KUKA KRL program: MyProgram_300().src

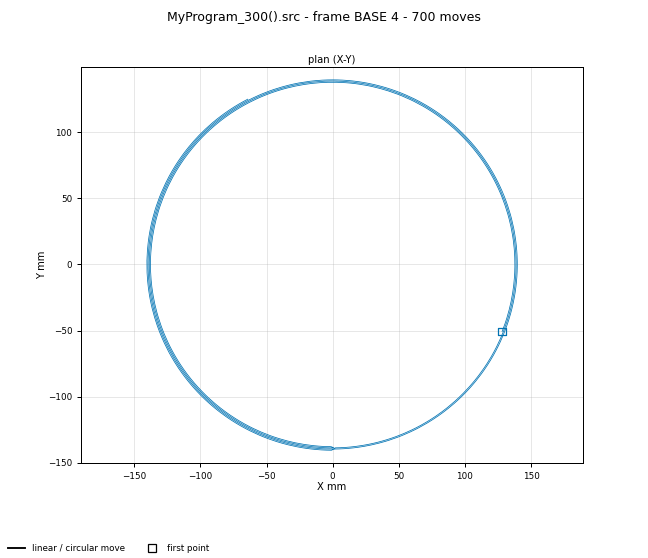
[picture p0: tool path of MyProgram_300().src in frame BASE 4, 700 of 700 moves have a stored position in this frame; points joined in program order, loops and branches not executed]
&ACCESS RVP
&REL 1
&PARAM TEMPLATE = C:\KRC\Roboter\Template\vorgabe
&PARAM EDITMASK = *
DEF MyProgram_300()
; ---- Setting reference (Base) ----
$BASE = BASE_DATA[4]

; --------------------------
; ---- Setting tool (TCP) ----
$TOOL = TOOL_DATA[3]
; --------------------------

$VEL.CP = VEL_APROX_PRINT
Startdeposition()
$VEL.CP = VEL_PRINT
LIN {X 128.1202,Y -50.7216,Z 179,A -18.2901,B 5.6421,C 0.2906,E1 5.7988,E2 470.655} C_DIS
LIN {X 129.3366,Y -47.5343,Z 179,A -16.9067,B 5.6423,C 0.2873,E1 5.8002,E2 469.2749} C_DIS
LIN {X 130.4678,Y -44.3354,Z 179,A -15.4081,B 5.6425,C 0.2821,E1 5.8015,E2 467.7637} C_DIS
LIN {X 131.6398,Y -40.7171,Z 179,A -13.99,B 5.6426,C 0.2803,E1 5.8027,E2 466.3653} C_DIS
LIN {X 132.591,Y -37.5041,Z 179,A -12.6322,B 5.6428,C 0.277,E1 5.8038,E2 465.0108} C_DIS
LIN {X 133.4585,Y -34.2894,Z 179,A -11.2835,B 5.643,C 0.2738,E1 5.8047,E2 463.6656} C_DIS
LIN {X 134.2751,Y -30.9365,Z 179,A -9.9543,B 5.643,C 0.2714,E1 5.8056,E2 462.3488} C_DIS
LIN {X 134.922,Y -27.9842,Z 179,A -8.7683,B 5.6432,C 0.269,E1 5.8063,E2 461.1708} C_DIS
LIN {X 135.5678,Y -24.6646,Z 179,A -7.2924,B 5.6434,C 0.264,E1 5.807,E2 459.6847} C_DIS
LIN {X 136.1099,Y -21.4723,Z 179,A -5.9815,B 5.6436,C 0.2607,E1 5.8076,E2 458.3773} C_DIS
LIN {X 136.5737,Y -18.2924,Z 179,A -4.6235,B 5.6438,C 0.2566,E1 5.8081,E2 457.0154} C_DIS
LIN {X 136.9237,Y -15.4683,Z 179,A -3.4321,B 5.6439,C 0.2531,E1 5.8085,E2 455.8221} C_DIS
LIN {X 137.2715,Y -11.9803,Z 179,A -2.254,B 5.6439,C 0.2533,E1 5.8088,E2 454.6786} C_DIS
LIN {X 137.5087,Y -8.8529,Z 179,A -0.9837,B 5.644,C 0.2502,E1 5.8091,E2 453.4116} C_DIS
LIN {X 137.658,Y -6.1429,Z 179,A 0.3699,B 5.6443,C 0.2434,E1 5.8093,E2 452.0283} C_DIS
LIN {X 137.7866,Y -1.5259,Z 179,A 2.0898,B 5.6444,C 0.2411,E1 5.8093,E2 450.3327} C_DIS
LIN {X 137.78,Y 1.9181,Z 179,A 3.3831,B 5.6445,C 0.2392,E1 5.8093,E2 449.056} C_DIS
LIN {X 137.7029,Y 4.993,Z 179,A 4.7743,B 5.6447,C 0.2338,E1 5.8093,E2 447.6496} C_DIS
LIN {X 137.58,Y 7.6943,Z 179,A 5.9871,B 5.6449,C 0.2292,E1 5.8091,E2 446.4246} C_DIS
LIN {X 137.2376,Y 12.3815,Z 179,A 7.8975,B 5.6451,C 0.2243,E1 5.8086,E2 444.5183} C_DIS
LIN {X 136.8687,Y 15.9359,Z 179,A 9.0863,B 5.6451,C 0.2248,E1 5.8083,E2 443.3665} C_DIS
LIN {X 136.5205,Y 18.6981,Z 179,A 10.364,B 5.6453,C 0.2196,E1 5.8078,E2 442.0727} C_DIS
LIN {X 136.0468,Y 21.8798,Z 179,A 11.6707,B 5.6454,C 0.2163,E1 5.8072,E2 440.7691} C_DIS
LIN {X 135.3992,Y 25.5723,Z 179,A 13.1704,B 5.6456,C 0.2129,E1 5.8065,E2 439.2758} C_DIS
LIN {X 134.7738,Y 28.6874,Z 179,A 14.4849,B 5.6457,C 0.2093,E1 5.8058,E2 437.9612} C_DIS
LIN {X 134.1493,Y 31.4869,Z 179,A 15.65,B 5.6458,C 0.2064,E1 5.805,E2 436.7989} C_DIS
LIN {X 133.3541,Y 34.7007,Z 179,A 17.1029,B 5.646,C 0.2014,E1 5.804,E2 435.3355} C_DIS
LIN {X 132.3654,Y 38.2933,Z 179,A 18.5158,B 5.646,C 0.1993,E1 5.803,E2 433.9389} C_DIS
LIN {X 131.3361,Y 41.6851,Z 179,A 19.9227,B 5.6462,C 0.1963,E1 5.8018,E2 432.5396} C_DIS
LIN {X 130.3079,Y 44.7966,Z 179,A 21.268,B 5.6462,C 0.1929,E1 5.8006,E2 431.1958} C_DIS
LIN {X 129.1837,Y 47.9425,Z 179,A 22.6404,B 5.6464,C 0.1895,E1 5.7993,E2 429.8246} C_DIS
LIN {X 127.9564,Y 51.1281,Z 179,A 24.0286,B 5.6465,C 0.1862,E1 5.7979,E2 428.4397} C_DIS
LIN {X 126.6436,Y 54.2982,Z 179,A 25.2652,B 5.6465,C 0.1854,E1 5.7966,E2 427.2263} C_DIS
LIN {X 125.23,Y 57.4833,Z 179,A 26.8315,B 5.6467,C 0.1798,E1 5.7948,E2 425.6445} C_DIS
LIN {X 123.762,Y 60.5793,Z 179,A 28.0749,B 5.6467,C 0.1789,E1 5.7933,E2 424.4233} C_DIS
LIN {X 122.1657,Y 63.7367,Z 179,A 29.6872,B 5.6469,C 0.173,E1 5.7912,E2 422.7925} C_DIS
LIN {X 120.2258,Y 67.3282,Z 179,A 31.3362,B 5.647,C 0.1695,E1 5.789,E2 421.1488} C_DIS
LIN {X 118.2543,Y 70.7336,Z 179,A 33.0192,B 5.6472,C 0.1648,E1 5.7866,E2 419.4592} C_DIS
LIN {X 115.8832,Y 74.555,Z 179,A 34.7836,B 5.6472,C 0.1619,E1 5.784,E2 417.7075} C_DIS
LIN {X 113.7346,Y 77.793,Z 179,A 36.4307,B 5.6474,C 0.1576,E1 5.7814,E2 416.0558} C_DIS
LIN {X 111.1958,Y 81.3807,Z 179,A 38.1794,B 5.6474,C 0.1546,E1 5.7786,E2 414.3164} C_DIS
LIN {X 108.6384,Y 84.7654,Z 179,A 39.9277,B 5.6476,C 0.1508,E1 5.7756,E2 412.5695} C_DIS
LIN {X 105.9924,Y 88.0508,Z 179,A 41.621,B 5.6476,C 0.1478,E1 5.7726,E2 410.8833} C_DIS
LIN {X 103.1924,Y 91.316,Z 179,A 43.4004,B 5.6477,C 0.1441,E1 5.7694,E2 409.1045} C_DIS
LIN {X 100.537,Y 94.2325,Z 179,A 45.056,B 5.6478,C 0.1404,E1 5.7662,E2 407.4466} C_DIS
LIN {X 97.4358,Y 97.4358,Z 179,A 46.8335,B 5.6478,C 0.1378,E1 5.7627,E2 405.6782} C_DIS
LIN {X 94.6416,Y 100.1512,Z 179,A 48.4576,B 5.648,C 0.1345,E1 5.7595,E2 404.0533} C_DIS
LIN {X 91.5999,Y 102.9413,Z 179,A 50.153,B 5.648,C 0.1315,E1 5.7559,E2 402.3603} C_DIS
LIN {X 88.2261,Y 105.8471,Z 179,A 51.9951,B 5.6481,C 0.1282,E1 5.752,E2 400.519} C_DIS
LIN {X 84.7654,Y 108.6384,Z 179,A 53.6964,B 5.6481,C 0.127,E1 5.7483,E2 398.836} C_DIS
LIN {X 81.5672,Y 111.0588,Z 179,A 55.3993,B 5.6482,C 0.1236,E1 5.7445,E2 397.1285} C_DIS
LIN {X 78.3355,Y 113.3623,Z 179,A 57.0178,B 5.6482,C 0.1214,E1 5.7408,E2 395.5139} C_DIS
LIN {X 74.8523,Y 115.6912,Z 179,A 58.7505,B 5.6483,C 0.1187,E1 5.7368,E2 393.7822} C_DIS
LIN {X 71.1191,Y 118.0229,Z 179,A 60.5116,B 5.6483,C 0.1169,E1 5.7326,E2 392.0298} C_DIS
LIN {X 67.896,Y 119.9067,Z 179,A 62.1383,B 5.6484,C 0.1137,E1 5.7286,E2 390.3937} C_DIS
LIN {X 64.437,Y 121.798,Z 179,A 63.6331,B 5.6484,C 0.1134,E1 5.725,E2 388.917} C_DIS
LIN {X 61.589,Y 123.2639,Z 179,A 64.888,B 5.6484,C 0.1127,E1 5.7219,E2 387.6718} C_DIS
LIN {X 58.6174,Y 124.7055,Z 179,A 66.4336,B 5.6485,C 0.1087,E1 5.718,E2 386.1049} C_DIS
LIN {X 54.9717,Y 126.3524,Z 179,A 67.7497,B 5.6485,C 0.1114,E1 5.7147,E2 384.832} C_DIS
LIN {X 52.3099,Y 127.48,Z 179,A 69.1382,B 5.6485,C 0.1075,E1 5.7111,E2 383.4206} C_DIS
LIN {X 49.1296,Y 128.7391,Z 179,A 70.6713,B 5.6486,C 0.1045,E1 5.707,E2 381.8739} C_DIS
LIN {X 45.4349,Y 130.0866,Z 179,A 71.9702,B 5.6486,C 0.1074,E1 5.7037,E2 380.6169} C_DIS
LIN {X 42.322,Y 131.1327,Z 179,A 73.5162,B 5.6486,C 0.1037,E1 5.6996,E2 379.0489} C_DIS
LIN {X 39.111,Y 132.1259,Z 179,A 74.9014,B 5.6486,C 0.1027,E1 5.6959,E2 377.6655} C_DIS
LIN {X 35.8968,Y 133.0352,Z 179,A 76.3077,B 5.6486,C 0.1014,E1 5.6921,E2 376.2573} C_DIS
LIN {X 32.6824,Y 133.8612,Z 179,A 77.4929,B 5.6486,C 0.1029,E1 5.6889,E2 375.0966} C_DIS
LIN {X 29.8812,Y 134.5161,Z 179,A 78.8355,B 5.6486,C 0.1002,E1 5.6852,E2 373.7363} C_DIS
LIN {X 26.6742,Y 135.1886,Z 179,A 80.3098,B 5.6487,C 0.098,E1 5.6812,E2 372.2485} C_DIS
LIN {X 22.9157,Y 135.874,Z 179,A 81.7673,B 5.6487,C 0.0988,E1 5.6772,E2 370.8077} C_DIS
LIN {X 19.8806,Y 136.3515,Z 179,A 83.0363,B 5.6487,C 0.0983,E1 5.6737,E2 369.5401} C_DIS
LIN {X 17.1127,Y 136.7283,Z 179,A 84.1924,B 5.6487,C 0.098,E1 5.6705,E2 368.3851} C_DIS
LIN {X 13.5516,Y 137.1253,Z 179,A 85.6745,B 5.6487,C 0.0975,E1 5.6664,E2 366.9045} C_DIS
LIN {X 10.1212,Y 137.4206,Z 179,A 87.0261,B 5.6487,C 0.0982,E1 5.6626,E2 365.5633} C_DIS
LIN {X 6.1429,Y 137.658,Z 179,A 88.8676,B 5.6487,C 0.0956,E1 5.6574,E2 363.6997} C_DIS
LIN {X 3.0585,Y 137.7611,Z 179,A 90.0316,B 5.6487,C 0.0969,E1 5.6542,E2 362.551} C_DIS
LIN {X -0.3905,Y 137.7929,Z 179,A 91.4644,B 5.6487,C 0.0969,E1 5.6502,E2 361.119} C_DIS
LIN {X -3.7662,Y 137.7414,Z 179,A 92.7926,B 5.6487,C 0.0978,E1 5.6466,E2 359.8007} C_DIS
LIN {X -6.5399,Y 137.6381,Z 179,A 93.8803,B 5.6487,C 0.0987,E1 5.6435,E2 358.7218} C_DIS
LIN {X -9.6512,Y 137.4549,Z 179,A 95.1792,B 5.6487,C 0.0989,E1 5.6399,E2 357.4232} C_DIS
LIN {X -12.9748,Y 137.1807,Z 179,A 96.6705,B 5.6487,C 0.0979,E1 5.6357,E2 355.9197} C_DIS
LIN {X -15.9359,Y 136.8687,Z 179,A 97.8121,B 5.6487,C 0.0994,E1 5.6326,E2 354.7906} C_DIS
LIN {X -19.278,Y 136.4376,Z 179,A 99.1541,B 5.6487,C 0.1006,E1 5.6289,E2 353.4567} C_DIS
LIN {X -21.8798,Y 136.0468,Z 179,A 100.4719,B 5.6487,C 0.0984,E1 5.6252,E2 352.112} C_DIS
LIN {X -25.4832,Y 135.4163,Z 179,A 102.0026,B 5.6487,C 0.099,E1 5.621,E2 350.5809} C_DIS
LIN {X -28.6874,Y 134.7738,Z 179,A 103.3702,B 5.6487,C 0.0996,E1 5.6172,E2 349.213} C_DIS
LIN {X -31.9883,Y 134.0285,Z 179,A 104.784,B 5.6487,C 0.1004,E1 5.6134,E2 347.7993} C_DIS
LIN {X -35.0817,Y 133.2525,Z 179,A 105.9762,B 5.6487,C 0.1028,E1 5.6102,E2 346.6243} C_DIS
LIN {X -37.9154,Y 132.476,Z 179,A 107.3552,B 5.6487,C 0.1019,E1 5.6065,E2 345.2268} C_DIS
LIN {X -41.3051,Y 131.4575,Z 179,A 108.9235,B 5.6487,C 0.102,E1 5.6022,E2 343.6474} C_DIS
LIN {X -44.745,Y 130.3258,Z 179,A 110.3596,B 5.6487,C 0.1041,E1 5.5985,E2 342.2209} C_DIS
LIN {X -47.9425,Y 129.1837,Z 179,A 111.7853,B 5.6486,C 0.1053,E1 5.5947,E2 340.7945} C_DIS
LIN {X -51.1281,Y 127.9564,Z 179,A 113.2197,B 5.6486,C 0.1066,E1 5.591,E2 339.3592} C_DIS
LIN {X -54.2982,Y 126.6436,Z 179,A 114.4971,B 5.6486,C 0.1098,E1 5.5878,E2 338.1013} C_DIS
LIN {X -57.4498,Y 125.2455,Z 179,A 116.1123,B 5.6486,C 0.1094,E1 5.5836,E2 336.4647} C_DIS
LIN {X -60.5793,Y 123.762,Z 179,A 117.4029,B 5.6484,C 0.1128,E1 5.5804,E2 335.1935} C_DIS
LIN {X -63.2885,Y 122.4011,Z 179,A 118.9792,B 5.6484,C 0.111,E1 5.5764,E2 333.5792} C_DIS
LIN {X -67.3282,Y 120.2258,Z 179,A 120.7792,B 5.6484,C 0.1147,E1 5.572,E2 331.7941} C_DIS
LIN {X -70.7933,Y 118.2187,Z 179,A 122.5502,B 5.6484,C 0.116,E1 5.5677,E2 330.0112} C_DIS
LIN {X -74.1106,Y 116.1677,Z 179,A 124.1123,B 5.6484,C 0.119,E1 5.564,E2 328.4577} C_DIS
LIN {X -77.4191,Y 113.9894,Z 179,A 125.8125,B 5.6483,C 0.121,E1 5.5601,E2 326.7522} C_DIS
LIN {X -80.5058,Y 111.8315,Z 179,A 127.3742,B 5.6483,C 0.1236,E1 5.5565,E2 325.1923} C_DIS
LIN {X -83.358,Y 109.722,Z 179,A 128.8729,B 5.6482,C 0.1259,E1 5.5532,E2 323.6919} C_DIS
LIN {X -86.6034,Y 107.1781,Z 179,A 130.6869,B 5.6482,C 0.1279,E1 5.5492,E2 321.867} C_DIS
LIN {X -89.9832,Y 104.3566,Z 179,A 132.5303,B 5.6481,C 0.1311,E1 5.5453,E2 320.0235} C_DIS
LIN {X -92.9238,Y 101.7479,Z 179,A 134.1412,B 5.648,C 0.1345,E1 5.5419,E2 318.4169} C_DIS
LIN {X -95.5258,Y 99.3091,Z 179,A 135.7639,B 5.648,C 0.1359,E1 5.5386,E2 316.7781} C_DIS
LIN {X -98.6888,Y 96.1665,Z 179,A 137.6469,B 5.6479,C 0.1394,E1 5.5349,E2 314.8931} C_DIS
LIN {X -101.7479,Y 92.9238,Z 179,A 139.4286,B 5.6477,C 0.144,E1 5.5315,E2 313.1219} C_DIS
LIN {X -104.1171,Y 90.2612,Z 179,A 140.9394,B 5.6477,C 0.1468,E1 5.5287,E2 311.6088} C_DIS
LIN {X -106.7267,Y 87.159,Z 179,A 142.7186,B 5.6476,C 0.1496,E1 5.5256,E2 309.8194} C_DIS
LIN {X -109.4793,Y 83.6753,Z 179,A 144.6009,B 5.6475,C 0.1534,E1 5.5223,E2 307.9342} C_DIS
LIN {X -112.1532,Y 80.0558,Z 179,A 146.5209,B 5.6474,C 0.1572,E1 5.5192,E2 306.0098} C_DIS
LIN {X -114.7454,Y 76.2943,Z 179,A 148.4151,B 5.6473,C 0.1618,E1 5.5162,E2 304.1179} C_DIS
LIN {X -116.7595,Y 73.1757,Z 179,A 149.9698,B 5.6472,C 0.1654,E1 5.5139,E2 302.5633} C_DIS
LIN {X -118.5889,Y 70.1722,Z 179,A 151.5732,B 5.6471,C 0.1676,E1 5.5116,E2 300.9434} C_DIS
LIN {X -120.8068,Y 66.2806,Z 179,A 153.4792,B 5.647,C 0.1718,E1 5.5089,E2 299.0336} C_DIS
LIN {X -122.6031,Y 62.8917,Z 179,A 154.8302,B 5.6468,C 0.1782,E1 5.5072,E2 297.7145} C_DIS
LIN {X -123.9586,Y 60.1808,Z 179,A 156.288,B 5.6468,C 0.1795,E1 5.5054,E2 296.2332} C_DIS
LIN {X -125.6114,Y 56.6453,Z 179,A 157.9691,B 5.6466,C 0.1832,E1 5.5034,E2 294.5461} C_DIS
LIN {X -126.9472,Y 53.5855,Z 179,A 159.2421,B 5.6465,C 0.1879,E1 5.5021,E2 293.2888} C_DIS
LIN {X -128.1202,Y 50.7216,Z 179,A 160.6856,B 5.6464,C 0.1898,E1 5.5005,E2 291.8269} C_DIS
LIN {X -129.3366,Y 47.5343,Z 179,A 162.1377,B 5.6463,C 0.1933,E1 5.4991,E2 290.3718} C_DIS
LIN {X -130.4678,Y 44.3354,Z 179,A 163.7124,B 5.6462,C 0.1956,E1 5.4977,E2 288.7778} C_DIS
LIN {X -131.6398,Y 40.7171,Z 179,A 165.2285,B 5.646,C 0.2005,E1 5.4964,E2 287.2712} C_DIS
LIN {X -132.591,Y 37.5041,Z 179,A 166.628,B 5.6459,C 0.2043,E1 5.4953,E2 285.8721} C_DIS
LIN {X -133.4585,Y 34.2894,Z 179,A 168.0458,B 5.6458,C 0.2078,E1 5.4943,E2 284.4513} C_DIS
LIN {X -134.1493,Y 31.4869,Z 179,A 169.3241,B 5.6457,C 0.2104,E1 5.4935,E2 283.1643} C_DIS
LIN {X -134.8625,Y 28.2769,Z 179,A 170.6761,B 5.6455,C 0.2144,E1 5.4927,E2 281.8154} C_DIS
LIN {X -135.5678,Y 24.6646,Z 179,A 172.2435,B 5.6454,C 0.2183,E1 5.4919,E2 280.2445} C_DIS
LIN {X -136.1099,Y 21.4723,Z 179,A 173.6384,B 5.6452,C 0.2216,E1 5.4912,E2 278.8446} C_DIS
LIN {X -136.5981,Y 18.1058,Z 179,A 175.0021,B 5.6451,C 0.2261,E1 5.4907,E2 277.4884} C_DIS
LIN {X -136.9766,Y 14.9766,Z 179,A 176.3733,B 5.6449,C 0.2293,E1 5.4903,E2 276.1107} C_DIS
LIN {X -137.2715,Y 11.9803,Z 179,A 177.545,B 5.6448,C 0.2336,E1 5.49,E2 274.9501} C_DIS
LIN {X -137.5087,Y 8.8529,Z 179,A 178.8823,B 5.6446,C 0.237,E1 5.4897,E2 273.6097} C_DIS
LIN {X -137.676,Y 5.6818,Z 179,A -179.5662,B 5.6446,C 0.2386,E1 5.4895,E2 272.0301} C_DIS
LIN {X -137.7757,Y 2.1767,Z 179,A -178.0739,B 5.6444,C 0.2424,E1 5.4894,E2 270.5345} C_DIS
LIN {X -137.78,Y -1.9181,Z 179,A -176.5203,B 5.6441,C 0.2487,E1 5.4894,E2 269.0012} C_DIS
LIN {X -137.7029,Y -4.993,Z 179,A -175.0548,B 5.6441,C 0.2506,E1 5.4895,E2 267.5131} C_DIS
LIN {X -137.5406,Y -8.3349,Z 179,A -173.6264,B 5.6439,C 0.2542,E1 5.4897,E2 266.0809} C_DIS
LIN {X -137.31,Y -11.5251,Z 179,A -172.3831,B 5.6437,C 0.2588,E1 5.49,E2 264.8496} C_DIS
LIN {X -137.0432,Y -14.3577,Z 179,A -171.0401,B 5.6436,C 0.2606,E1 5.4904,E2 263.4872} C_DIS
LIN {X -136.7283,Y -17.1127,Z 179,A -169.8549,B 5.6434,C 0.2636,E1 5.4908,E2 262.2987} C_DIS
LIN {X -136.2166,Y -20.7832,Z 179,A -168.2945,B 5.6432,C 0.2677,E1 5.4914,E2 260.7369} C_DIS
LIN {X -135.7188,Y -23.8206,Z 179,A -166.937,B 5.6432,C 0.2706,E1 5.492,E2 259.3704} C_DIS
LIN {X -135.1051,Y -27.0843,Z 179,A -165.5365,B 5.6429,C 0.2742,E1 5.4928,E2 257.9684} C_DIS
LIN {X -134.4222,Y -30.2921,Z 179,A -164.2114,B 5.6427,C 0.2784,E1 5.4936,E2 256.6491} C_DIS
LIN {X -133.7621,Y -33.0935,Z 179,A -162.9068,B 5.6427,C 0.2807,E1 5.4944,E2 255.3315} C_DIS
LIN {X -132.9255,Y -36.3081,Z 179,A -161.4887,B 5.6424,C 0.2841,E1 5.4955,E2 253.9096} C_DIS
LIN {X -132.0055,Y -39.5222,Z 179,A -159.9761,B 5.6424,C 0.2867,E1 5.4967,E2 252.3821} C_DIS
LIN {X -130.8244,Y -43.2644,Z 179,A -158.4218,B 5.6421,C 0.2918,E1 5.498,E2 250.8386} C_DIS
LIN {X -129.7654,Y -46.3451,Z 179,A -156.9967,B 5.6419,C 0.2947,E1 5.4993,E2 249.4052} C_DIS
LIN {X -128.5807,Y -49.537,Z 179,A -155.5445,B 5.6417,C 0.2981,E1 5.5008,E2 247.9493} C_DIS
LIN {X -127.3107,Y -52.7153,Z 179,A -154.0856,B 5.6415,C 0.3015,E1 5.5023,E2 246.4865} C_DIS
LIN {X -125.9222,Y -55.9503,Z 179,A -152.6076,B 5.6414,C 0.3051,E1 5.504,E2 245.0074} C_DIS
LIN {X -124.5144,Y -59.0175,Z 179,A -151.1192,B 5.6412,C 0.3079,E1 5.5057,E2 243.5089} C_DIS
LIN {X -123.0196,Y -62.0736,Z 179,A -149.8193,B 5.6409,C 0.3126,E1 5.5073,E2 242.2244} C_DIS
LIN {X -121.2832,Y -65.4041,Z 179,A -148.0153,B 5.6409,C 0.314,E1 5.5097,E2 240.39} C_DIS
LIN {X -119.3602,Y -68.851,Z 179,A -146.3393,B 5.6407,C 0.3177,E1 5.512,E2 238.7102} C_DIS
LIN {X -117.1055,Y -72.6196,Z 179,A -144.4629,B 5.6404,C 0.3216,E1 5.5148,E2 236.8281} C_DIS
LIN {X -114.8485,Y -76.14,Z 179,A -142.7104,B 5.6402,C 0.3255,E1 5.5175,E2 235.0745} C_DIS
LIN {X -112.4719,Y -79.6078,Z 179,A -140.9621,B 5.64,C 0.3295,E1 5.5202,E2 233.3268} C_DIS
LIN {X -110.1198,Y -82.8308,Z 179,A -139.1932,B 5.6398,C 0.3321,E1 5.5232,E2 231.5443} C_DIS
LIN {X -107.393,Y -86.3369,Z 179,A -137.3171,B 5.6396,C 0.3358,E1 5.5265,E2 229.665} C_DIS
LIN {X -104.5496,Y -89.7591,Z 179,A -135.5239,B 5.6393,C 0.3403,E1 5.5297,E2 227.8797} C_DIS
LIN {X -101.9011,Y -92.7549,Z 179,A -133.8008,B 5.6392,C 0.3431,E1 5.5329,E2 226.1493} C_DIS
LIN {X -98.9435,Y -95.9034,Z 179,A -131.9483,B 5.639,C 0.346,E1 5.5365,E2 224.2899} C_DIS
LIN {X -96.0025,Y -98.8475,Z 179,A -130.2391,B 5.6388,C 0.3496,E1 5.5399,E2 222.5839} C_DIS
LIN {X -93.4122,Y -101.299,Z 179,A -128.6366,B 5.6387,C 0.3511,E1 5.5432,E2 220.9661} C_DIS
LIN {X -90.2612,Y -104.1171,Z 179,A -126.9441,B 5.6384,C 0.355,E1 5.5467,E2 219.2824} C_DIS
LIN {X -87.5408,Y -106.4147,Z 179,A -125.3836,B 5.6384,C 0.3567,E1 5.5501,E2 217.7118} C_DIS
LIN {X -84.2429,Y -109.0433,Z 179,A -123.6318,B 5.6381,C 0.3596,E1 5.5539,E2 215.9604} C_DIS
LIN {X -81.0398,Y -111.4445,Z 179,A -121.9719,B 5.638,C 0.3624,E1 5.5577,E2 214.3012} C_DIS
LIN {X -77.665,Y -113.8225,Z 179,A -120.1362,B 5.6379,C 0.3637,E1 5.5619,E2 212.4501} C_DIS
LIN {X -73.9206,Y -116.2894,Z 179,A -118.3438,B 5.6377,C 0.3672,E1 5.5661,E2 210.6671} C_DIS
LIN {X -70.7336,Y -118.2543,Z 179,A -116.67,B 5.6377,C 0.368,E1 5.5701,E2 208.9781} C_DIS
LIN {X -67.0507,Y -120.3811,Z 179,A -114.9488,B 5.6374,C 0.3709,E1 5.5743,E2 207.2631} C_DIS
LIN {X -63.2885,Y -122.4011,Z 179,A -113.1863,B 5.6373,C 0.3732,E1 5.5787,E2 205.5021} C_DIS
LIN {X -60.1808,Y -123.9586,Z 179,A -111.581,B 5.6373,C 0.373,E1 5.5827,E2 203.8759} C_DIS
LIN {X -56.5777,Y -125.6416,Z 179,A -110.2501,B 5.6369,C 0.3785,E1 5.586,E2 202.5869} C_DIS
LIN {X -53.894,Y -126.8184,Z 179,A -108.8301,B 5.6369,C 0.3774,E1 5.5897,E2 201.1405} C_DIS
LIN {X -50.327,Y -128.2736,Z 179,A -107.1925,B 5.6369,C 0.3785,E1 5.594,E2 199.4979} C_DIS
LIN {X -47.5343,Y -129.3366,Z 179,A -105.9653,B 5.6369,C 0.3798,E1 5.5972,E2 198.2726} C_DIS
LIN {X -44.3354,Y -130.4678,Z 179,A -104.4185,B 5.6369,C 0.3794,E1 5.6013,E2 196.7077} C_DIS
LIN {X -40.7171,Y -131.6398,Z 179,A -102.9559,B 5.6367,C 0.3819,E1 5.6052,E2 195.2603} C_DIS
LIN {X -37.4292,Y -132.612,Z 179,A -101.516,B 5.6367,C 0.3827,E1 5.609,E2 193.8181} C_DIS
LIN {X -34.2894,Y -133.4585,Z 179,A -100.166,B 5.6366,C 0.3836,E1 5.6127,E2 192.4681} C_DIS
LIN {X -31.4869,Y -134.1493,Z 179,A -98.9611,B 5.6366,C 0.3842,E1 5.616,E2 191.2624} C_DIS
LIN {X -28.2769,Y -134.8625,Z 179,A -97.4349,B 5.6366,C 0.3829,E1 5.6202,E2 189.7149} C_DIS
LIN {X -24.6646,Y -135.5678,Z 179,A -96.0569,B 5.6365,C 0.3854,E1 5.6239,E2 188.3563} C_DIS
LIN {X -21.4723,Y -136.1099,Z 179,A -94.7086,B 5.6365,C 0.3858,E1 5.6276,E2 187.0074} C_DIS
LIN {X -18.2924,Y -136.5737,Z 179,A -93.5219,B 5.6363,C 0.388,E1 5.6309,E2 185.8397} C_DIS
LIN {X -15.0053,Y -136.9735,Z 179,A -91.9626,B 5.6364,C 0.386,E1 5.6353,E2 184.256} C_DIS
LIN {X -10.8138,Y -137.37,Z 179,A -90.1274,B 5.6364,C 0.3852,E1 5.6404,E2 182.4091} C_DIS
LIN {X -7.6943,Y -137.58,Z 179,A -88.946,B 5.6364,C 0.3868,E1 5.6437,E2 181.2427} C_DIS
LIN {X -4.2037,Y -137.7292,Z 179,A -87.6415,B 5.6362,C 0.3886,E1 5.6472,E2 179.957} C_DIS
LIN {X -1.2026,Y -137.7884,Z 179,A -86.1996,B 5.6364,C 0.386,E1 5.6513,E2 178.4891} C_DIS
LIN {X -1.2026,Y -137.7884,Z 179,A -86.1996,B 5.6364,C 0.386,E1 5.6513,E2 178.4891} C_DIS
Enddeposition()
LIN {X 0.9856,Y -138.6883,Z 179,A -85.6514,B 5.6021,C 0.3933,E1 5.6189,E2 178.0298} C_DIS
Startdeposition()
$VEL.CP = VEL_PRINT
LIN {X -2.3795,Y -138.6758,Z 179,A -87.2968,B 5.6019,C 0.3968,E1 5.6142,E2 179.7096} C_DIS
LIN {X -6.0242,Y -138.5667,Z 179,A -88.891,B 5.6019,C 0.3979,E1 5.6097,E2 181.316} C_DIS
LIN {X -9.7456,Y -138.3538,Z 179,A -90.413,B 5.6019,C 0.3976,E1 5.6055,E2 182.8363} C_DIS
LIN {X -14.0264,Y -137.9872,Z 179,A -92.1915,B 5.6019,C 0.3974,E1 5.6006,E2 184.6159} C_DIS
LIN {X -17.9699,Y -137.527,Z 179,A -93.7461,B 5.6019,C 0.396,E1 5.5963,E2 186.1599} C_DIS
LIN {X -21.384,Y -137.0377,Z 179,A -95.0296,B 5.6021,C 0.3938,E1 5.5928,E2 187.4254} C_DIS
LIN {X -26.6137,Y -136.1199,Z 179,A -97.2944,B 5.6021,C 0.3938,E1 5.5865,E2 189.7004} C_DIS
LIN {X -34.3932,Y -134.3642,Z 179,A -100.8331,B 5.602,C 0.3951,E1 5.5768,E2 193.272} C_DIS
LIN {X -38.5546,Y -133.2301,Z 179,A -102.354,B 5.6023,C 0.3908,E1 5.5728,E2 194.7593} C_DIS
LIN {X -42.0759,Y -132.1596,Z 179,A -104.0679,B 5.6023,C 0.392,E1 5.5682,E2 196.4988} C_DIS
LIN {X -46.1855,Y -130.7824,Z 179,A -106.112,B 5.6021,C 0.3935,E1 5.5627,E2 198.5763} C_DIS
LIN {X -49.2387,Y -129.6628,Z 179,A -107.3125,B 5.6023,C 0.3907,E1 5.5596,E2 199.7584} C_DIS
LIN {X -53.4297,Y -127.9912,Z 179,A -109.0334,B 5.6025,C 0.3872,E1 5.5552,E2 201.4609} C_DIS
LIN {X -58.9396,Y -125.5517,Z 179,A -112.5014,B 5.602,C 0.3957,E1 5.5461,E2 205.0558} C_DIS
LIN {X -64.9557,Y -122.5459,Z 179,A -114.3398,B 5.6029,C 0.3817,E1 5.5418,E2 206.773} C_DIS
LIN {X -68.3132,Y -120.7084,Z 179,A -116.0962,B 5.6029,C 0.3817,E1 5.5375,E2 208.5522} C_DIS
LIN {X -72.0687,Y -118.5043,Z 179,A -117.8743,B 5.6031,C 0.379,E1 5.5332,E2 210.3277} C_DIS
LIN {X -76.1971,Y -115.8924,Z 179,A -119.93,B 5.6033,C 0.3765,E1 5.5284,E2 212.3882} C_DIS
LIN {X -78.8038,Y -114.1366,Z 179,A -122.0735,B 5.6028,C 0.3837,E1 5.5232,E2 214.6405} C_DIS
LIN {X -84.1719,Y -110.2367,Z 179,A -124.0371,B 5.6036,C 0.3709,E1 5.519,E2 216.5039} C_DIS
LIN {X -87.8184,Y -107.3544,Z 179,A -125.9821,B 5.6038,C 0.3679,E1 5.5148,E2 218.4519} C_DIS
LIN {X -91.3324,Y -104.3813,Z 179,A -127.8877,B 5.6041,C 0.3646,E1 5.5108,E2 220.3578} C_DIS
LIN {X -94.5984,Y -101.4307,Z 179,A -129.7407,B 5.6043,C 0.3616,E1 5.5069,E2 222.2149} C_DIS
LIN {X -97.9095,Y -98.2385,Z 179,A -131.7023,B 5.6044,C 0.3586,E1 5.503,E2 224.1841} C_DIS
LIN {X -101.1384,Y -94.9115,Z 179,A -133.6563,B 5.6047,C 0.3552,E1 5.4992,E2 226.1426} C_DIS
LIN {X -104.1118,Y -91.6399,Z 179,A -135.5186,B 5.6049,C 0.3518,E1 5.4957,E2 228.0091} C_DIS
LIN {X -107.1066,Y -88.1215,Z 179,A -137.4629,B 5.6051,C 0.3481,E1 5.4923,E2 229.9574} C_DIS
LIN {X -109.8719,Y -84.6485,Z 179,A -139.0725,B 5.6055,C 0.3418,E1 5.4895,E2 231.5375} C_DIS
LIN {X -112.3797,Y -81.2887,Z 179,A -141.0873,B 5.6055,C 0.3408,E1 5.4861,E2 233.5881} C_DIS
LIN {X -115.0488,Y -77.4657,Z 179,A -143.0067,B 5.6058,C 0.3363,E1 5.4831,E2 235.506} C_DIS
LIN {X -117.3652,Y -73.9085,Z 179,A -144.8304,B 5.606,C 0.3329,E1 5.4803,E2 237.3379} C_DIS
LIN {X -119.7517,Y -69.9763,Z 179,A -146.7914,B 5.6063,C 0.3289,E1 5.4775,E2 239.3059} C_DIS
LIN {X -122.6672,Y -64.7248,Z 179,A -149.2164,B 5.6066,C 0.3223,E1 5.4743,E2 241.7225} C_DIS
LIN {X -124.267,Y -61.5976,Z 179,A -150.7321,B 5.6068,C 0.3192,E1 5.4723,E2 243.2457} C_DIS
LIN {X -125.6409,Y -58.7468,Z 179,A -152.1122,B 5.607,C 0.3166,E1 5.4707,E2 244.6346} C_DIS
LIN {X -127.1882,Y -55.3148,Z 179,A -153.6822,B 5.6072,C 0.3128,E1 5.4689,E2 246.2056} C_DIS
LIN {X -128.4935,Y -52.2117,Z 179,A -154.902,B 5.6075,C 0.3075,E1 5.4676,E2 247.4028} C_DIS
LIN {X -129.7664,Y -48.9622,Z 179,A -156.3596,B 5.6077,C 0.3039,E1 5.4662,E2 248.8617} C_DIS
LIN {X -131.2255,Y -44.9076,Z 179,A -158.4882,B 5.6077,C 0.3025,E1 5.4641,E2 251.0339} C_DIS
LIN {X -132.5037,Y -40.9813,Z 179,A -160.0567,B 5.6081,C 0.2966,E1 5.4628,E2 252.5838} C_DIS
LIN {X -133.506,Y -37.5863,Z 179,A -161.6729,B 5.6081,C 0.294,E1 5.4615,E2 254.2187} C_DIS
LIN {X -134.3506,Y -34.4467,Z 179,A -163.0292,B 5.6084,C 0.2905,E1 5.4606,E2 255.5759} C_DIS
LIN {X -135.1642,Y -31.1004,Z 179,A -164.4863,B 5.6086,C 0.2869,E1 5.4596,E2 257.0365} C_DIS
LIN {X -135.8316,Y -28.0443,Z 179,A -165.7434,B 5.6088,C 0.283,E1 5.4589,E2 258.2882} C_DIS
LIN {X -136.4427,Y -24.9036,Z 179,A -167.1729,B 5.6088,C 0.2803,E1 5.4582,E2 259.7306} C_DIS
LIN {X -137.0378,Y -21.3833,Z 179,A -168.6708,B 5.6091,C 0.2764,E1 5.4575,E2 261.2304} C_DIS
LIN {X -137.5408,Y -17.8642,Z 179,A -170.1694,B 5.6093,C 0.2725,E1 5.4569,E2 262.7317} C_DIS
LIN {X -137.9188,Y -14.6638,Z 179,A -171.5871,B 5.6094,C 0.2696,E1 5.4565,E2 264.1595} C_DIS
LIN {X -138.3065,Y -10.3931,Z 179,A -173.3571,B 5.6097,C 0.2645,E1 5.4561,E2 265.9279} C_DIS
LIN {X -138.521,Y -6.9683,Z 179,A -174.8543,B 5.6098,C 0.2612,E1 5.4558,E2 267.4342} C_DIS
LIN {X -138.6383,Y -4.012,Z 179,A -176.196,B 5.6099,C 0.2589,E1 5.4558,E2 268.79} C_DIS
LIN {X -138.6875,Y 1.6755,Z 179,A -178.5572,B 5.6102,C 0.2523,E1 5.4558,E2 271.151} C_DIS
LIN {X -138.595,Y 5.2983,Z 179,A 179.9546,B 5.6104,C 0.2479,E1 5.4558,E2 272.6368} C_DIS
LIN {X -138.379,Y 9.4003,Z 179,A 177.8743,B 5.6104,C 0.2466,E1 5.4562,E2 274.7639} C_DIS
LIN {X -138.09,Y 12.9551,Z 179,A 176.5721,B 5.6107,C 0.2409,E1 5.4565,E2 276.0435} C_DIS
LIN {X -137.577,Y 17.5883,Z 179,A 174.703,B 5.611,C 0.2349,E1 5.4572,E2 277.904} C_DIS
LIN {X -137.1594,Y 20.5978,Z 179,A 173.338,B 5.611,C 0.2324,E1 5.4577,E2 279.2817} C_DIS
LIN {X -136.4505,Y 24.86,Z 179,A 171.2437,B 5.6112,C 0.2302,E1 5.4588,E2 281.4133} C_DIS
LIN {X -135.7088,Y 28.6371,Z 179,A 169.9498,B 5.6115,C 0.223,E1 5.4595,E2 282.6688} C_DIS
LIN {X -134.9647,Y 31.9591,Z 179,A 168.6744,B 5.6117,C 0.2179,E1 5.4602,E2 283.9266} C_DIS
LIN {X -134.0575,Y 35.5691,Z 179,A 167.0236,B 5.6117,C 0.2147,E1 5.4614,E2 285.5902} C_DIS
LIN {X -133.2428,Y 38.5113,Z 179,A 165.6366,B 5.6119,C 0.2124,E1 5.4625,E2 286.9919} C_DIS
LIN {X -132.1578,Y 42.0815,Z 179,A 164.1431,B 5.612,C 0.2077,E1 5.4637,E2 288.4781} C_DIS
LIN {X -131.1591,Y 45.0991,Z 179,A 162.4429,B 5.612,C 0.2077,E1 5.4653,E2 290.2254} C_DIS
LIN {X -129.8963,Y 48.6153,Z 179,A 160.4975,B 5.612,C 0.2073,E1 5.4672,E2 292.2193} C_DIS
LIN {X -127.9288,Y 53.5792,Z 179,A 158.9136,B 5.6125,C 0.1957,E1 5.4688,E2 293.7241} C_DIS
LIN {X -126.4742,Y 56.9285,Z 179,A 157.2879,B 5.6125,C 0.1929,E1 5.4707,E2 295.3631} C_DIS
LIN {X -124.6171,Y 60.8878,Z 179,A 155.4608,B 5.6127,C 0.1884,E1 5.4729,E2 297.1912} C_DIS
LIN {X -121.6234,Y 66.6699,Z 179,A 152.6675,B 5.6129,C 0.1826,E1 5.4765,E2 299.995} C_DIS
LIN {X -119.3839,Y 70.6023,Z 179,A 150.7415,B 5.613,C 0.1786,E1 5.4792,E2 301.9264} C_DIS
LIN {X -117.101,Y 74.3271,Z 179,A 148.9312,B 5.6132,C 0.1743,E1 5.4819,E2 303.7358} C_DIS
LIN {X -114.633,Y 78.0799,Z 179,A 147.0189,B 5.6132,C 0.1704,E1 5.4849,E2 305.6535} C_DIS
LIN {X -112.0391,Y 81.7587,Z 179,A 145.2417,B 5.6134,C 0.1653,E1 5.4878,E2 307.4189} C_DIS
LIN {X -109.7097,Y 84.8578,Z 179,A 143.4742,B 5.6135,C 0.1633,E1 5.4908,E2 309.2056} C_DIS
LIN {X -106.8756,Y 88.4005,Z 179,A 141.6211,B 5.6136,C 0.1589,E1 5.494,E2 311.0544} C_DIS
LIN {X -104.1404,Y 91.6075,Z 179,A 140.0852,B 5.6138,C 0.1532,E1 5.4968,E2 312.5634} C_DIS
LIN {X -102.4541,Y 93.4898,Z 179,A 138.619,B 5.6138,C 0.1551,E1 5.4996,E2 314.081} C_DIS
LIN {X -98.8812,Y 97.2604,Z 179,A 136.6114,B 5.6138,C 0.1494,E1 5.5035,E2 316.0696} C_DIS
LIN {X -96.0041,Y 100.1014,Z 179,A 134.8881,B 5.614,C 0.1466,E1 5.5069,E2 317.798} C_DIS
LIN {X -92.5867,Y 103.2702,Z 179,A 132.8023,B 5.614,C 0.1445,E1 5.5113,E2 319.9021} C_DIS
LIN {X -88.7886,Y 106.5542,Z 179,A 130.7405,B 5.6141,C 0.1406,E1 5.5157,E2 321.9607} C_DIS
LIN {X -85.5317,Y 109.1851,Z 179,A 129.0853,B 5.6142,C 0.1368,E1 5.5193,E2 323.6052} C_DIS
LIN {X -82.3707,Y 111.5893,Z 179,A 127.2515,B 5.6142,C 0.136,E1 5.5234,E2 325.4615} C_DIS
LIN {X -78.1677,Y 114.5731,Z 179,A 125.1757,B 5.6143,C 0.132,E1 5.5282,E2 327.5291} C_DIS
LIN {X -74.3457,Y 117.0892,Z 179,A 123.2345,B 5.6143,C 0.1297,E1 5.5327,E2 329.4751} C_DIS
LIN {X -70.3761,Y 119.5168,Z 179,A 121.3109,B 5.6144,C 0.1269,E1 5.5373,E2 331.3973} C_DIS
LIN {X -66.2216,Y 121.8679,Z 179,A 119.3421,B 5.6145,C 0.1242,E1 5.5421,E2 333.3642} C_DIS
LIN {X -62.9011,Y 123.612,Z 179,A 118.0695,B 5.6146,C 0.1192,E1 5.5452,E2 334.6014} C_DIS
LIN {X -58.2782,Y 125.8576,Z 179,A 115.7344,B 5.6146,C 0.119,E1 5.5511,E2 336.9612} C_DIS
LIN {X -55.481,Y 127.1164,Z 179,A 113.6914,B 5.6145,C 0.126,E1 5.5566,E2 339.0983} C_DIS
LIN {X -50.2571,Y 129.27,Z 179,A 112.1369,B 5.6147,C 0.1151,E1 5.5604,E2 340.5559} C_DIS
LIN {X -47.2419,Y 130.4023,Z 179,A 110.7576,B 5.6147,C 0.1143,E1 5.564,E2 341.9403} C_DIS
LIN {X -44.1677,Y 131.4757,Z 179,A 109.3415,B 5.6147,C 0.1139,E1 5.5678,E2 343.3642} C_DIS
LIN {X -40.74,Y 132.5775,Z 179,A 107.8429,B 5.6147,C 0.1128,E1 5.5718,E2 344.8632} C_DIS
LIN {X -37.8856,Y 133.4223,Z 179,A 106.5569,B 5.6147,C 0.1125,E1 5.5752,E2 346.1554} C_DIS
LIN {X -34.3789,Y 134.3678,Z 179,A 105.105,B 5.6147,C 0.1109,E1 5.5791,E2 347.6004} C_DIS
LIN {X -31.4816,Y 135.0771,Z 179,A 103.7871,B 5.6147,C 0.1112,E1 5.5828,E2 348.9282} C_DIS
LIN {X -28.2843,Y 135.7828,Z 179,A 102.6054,B 5.6148,C 0.1084,E1 5.5859,E2 350.088} C_DIS
LIN {X -24.4077,Y 136.5314,Z 179,A 100.9256,B 5.6148,C 0.1082,E1 5.5906,E2 351.7728} C_DIS
LIN {X -21.0653,Y 137.087,Z 179,A 99.3529,B 5.6148,C 0.1096,E1 5.5949,E2 353.3661} C_DIS
LIN {X -17.3651,Y 137.6063,Z 179,A 97.8178,B 5.6148,C 0.109,E1 5.5992,E2 354.8994} C_DIS
LIN {X -12.5547,Y 138.1285,Z 179,A 95.7735,B 5.6148,C 0.109,E1 5.6049,E2 356.9482} C_DIS
LIN {X -6.081,Y 138.5645,Z 179,A 93.1395,B 5.6148,C 0.1081,E1 5.6122,E2 359.5753} C_DIS
LIN {X -2.2055,Y 138.6787,Z 179,A 91.6845,B 5.6148,C 0.1063,E1 5.6162,E2 361.0115} C_DIS
LIN {X 1.2114,Y 138.6917,Z 179,A 90.2148,B 5.6148,C 0.1071,E1 5.6204,E2 362.4877} C_DIS
LIN {X 5.3909,Y 138.5914,Z 179,A 88.5576,B 5.6148,C 0.1064,E1 5.625,E2 364.1355} C_DIS
LIN {X 8.5585,Y 138.4318,Z 179,A 87.1852,B 5.6148,C 0.1075,E1 5.6288,E2 365.5151} C_DIS
LIN {X 12.7647,Y 138.1083,Z 179,A 85.4617,B 5.6148,C 0.1077,E1 5.6336,E2 367.2356} C_DIS
LIN {X 15.4238,Y 137.837,Z 179,A 83.4439,B 5.6146,C 0.1195,E1 5.6395,E2 369.3648} C_DIS
LIN {X 22.1229,Y 136.9221,Z 179,A 81.5072,B 5.6148,C 0.1101,E1 5.6446,E2 371.1961} C_DIS
LIN {X 25.2387,Y 136.3827,Z 179,A 79.5311,B 5.6146,C 0.1193,E1 5.6502,E2 373.2539} C_DIS
LIN {X 30.828,Y 135.2264,Z 179,A 77.64,B 5.6147,C 0.1149,E1 5.6552,E2 375.0872} C_DIS
LIN {X 34.0788,Y 134.4439,Z 179,A 76.5912,B 5.6147,C 0.1116,E1 5.6579,E2 376.0947} C_DIS
LIN {X 36.9019,Y 133.6974,Z 179,A 75.4935,B 5.6147,C 0.1111,E1 5.6609,E2 377.1787} C_DIS
LIN {X 40.2012,Y 132.7424,Z 179,A 73.8778,B 5.6147,C 0.1149,E1 5.6653,E2 378.8186} C_DIS
LIN {X 43.6957,Y 131.6329,Z 179,A 72.4424,B 5.6147,C 0.1152,E1 5.669,E2 380.2438} C_DIS
LIN {X 46.6657,Y 130.61,Z 179,A 71.1344,B 5.6147,C 0.1166,E1 5.6725,E2 381.5529} C_DIS
LIN {X 50.2422,Y 129.2758,Z 179,A 69.6266,B 5.6147,C 0.1173,E1 5.6764,E2 383.0519} C_DIS
LIN {X 53.0207,Y 128.162,Z 179,A 68.1984,B 5.6146,C 0.1213,E1 5.6802,E2 384.5037} C_DIS
LIN {X 56.3593,Y 126.7289,Z 179,A 66.2506,B 5.6144,C 0.129,E1 5.6853,E2 386.5063} C_DIS
LIN {X 61.1421,Y 124.4917,Z 179,A 64.9225,B 5.6146,C 0.1203,E1 5.6884,E2 387.729} C_DIS
LIN {X 64.1195,Y 122.9851,Z 179,A 63.3541,B 5.6145,C 0.1247,E1 5.6923,E2 389.321} C_DIS
LIN {X 68.08,Y 120.8394,Z 179,A 61.4852,B 5.6145,C 0.1274,E1 5.6969,E2 391.1909} C_DIS
LIN {X 71.9409,Y 118.5816,Z 179,A 59.5585,B 5.6143,C 0.1312,E1 5.7015,E2 393.1274} C_DIS
LIN {X 76.0047,Y 116.019,Z 179,A 56.922,B 5.614,C 0.1434,E1 5.7079,E2 395.8444} C_DIS
LIN {X 81.2379,Y 112.4165,Z 179,A 55.0737,B 5.6142,C 0.1369,E1 5.7119,E2 397.5971} C_DIS
LIN {X 84.7522,Y 109.7915,Z 179,A 53.2839,B 5.6142,C 0.1398,E1 5.7158,E2 399.3844} C_DIS
LIN {X 88.3614,Y 106.9079,Z 179,A 51.408,B 5.6141,C 0.1428,E1 5.7199,E2 401.2565} C_DIS
LIN {X 91.8069,Y 103.9641,Z 179,A 49.6228,B 5.6141,C 0.145,E1 5.7236,E2 403.0312} C_DIS
LIN {X 94.0924,Y 101.9007,Z 179,A 48.3063,B 5.6139,C 0.1482,E1 5.7264,E2 404.3535} C_DIS
LIN {X 97.9706,Y 98.1778,Z 179,A 46.1505,B 5.6139,C 0.1517,E1 5.7307,E2 406.5017} C_DIS
LIN {X 100.9064,Y 95.1574,Z 179,A 44.4439,B 5.6137,C 0.1548,E1 5.734,E2 408.2045} C_DIS
LIN {X 104.0039,Y 91.7618,Z 179,A 42.5816,B 5.6137,C 0.1583,E1 5.7374,E2 410.0627} C_DIS
LIN {X 106.8839,Y 88.3905,Z 179,A 40.6721,B 5.6135,C 0.1634,E1 5.7409,E2 411.9825} C_DIS
LIN {X 110.0628,Y 84.3993,Z 179,A 38.7021,B 5.6135,C 0.1661,E1 5.7442,E2 413.936} C_DIS
LIN {X 112.83,Y 80.6624,Z 179,A 36.8898,B 5.6133,C 0.169,E1 5.7472,E2 415.7354} C_DIS
LIN {X 115.139,Y 77.3317,Z 179,A 35.0792,B 5.6132,C 0.1749,E1 5.7501,E2 417.5637} C_DIS
LIN {X 117.3178,Y 73.9836,Z 179,A 32.4923,B 5.6126,C 0.1929,E1 5.7541,E2 420.2676} C_DIS
LIN {X 121.5463,Y 66.8111,Z 179,A 30.1892,B 5.6129,C 0.1844,E1 5.757,E2 422.431} C_DIS
LIN {X 123.4156,Y 63.2868,Z 179,A 28.8534,B 5.6129,C 0.1839,E1 5.7587,E2 423.7282} C_DIS
LIN {X 124.9892,Y 60.1191,Z 179,A 26.9352,B 5.6125,C 0.1945,E1 5.7611,E2 425.7046} C_DIS
LIN {X 126.5752,Y 56.7029,Z 179,A 24.3987,B 5.6118,C 0.2133,E1 5.7641,E2 428.3639} C_DIS
LIN {X 130.0918,Y 48.0935,Z 179,A 21.8922,B 5.6122,C 0.2034,E1 5.7665,E2 430.706} C_DIS
LIN {X 131.5044,Y 44.0815,Z 179,A 20.2798,B 5.6122,C 0.2059,E1 5.7679,E2 432.3011} C_DIS
LIN {X 132.5753,Y 40.7474,Z 179,A 18.8829,B 5.612,C 0.209,E1 5.7691,E2 433.6926} C_DIS
LIN {X 133.5246,Y 37.5198,Z 179,A 17.5292,B 5.6119,C 0.2123,E1 5.7701,E2 435.0425} C_DIS
LIN {X 134.409,Y 34.2166,Z 179,A 16.0616,B 5.6117,C 0.217,E1 5.7711,E2 436.518} C_DIS
LIN {X 135.3608,Y 30.2397,Z 179,A 14.5284,B 5.6117,C 0.2193,E1 5.7721,E2 438.0325} C_DIS
LIN {X 136.3838,Y 25.2324,Z 179,A 12.2871,B 5.6113,C 0.2272,E1 5.7733,E2 440.2918} C_DIS
LIN {X 137.5625,Y 17.6992,Z 179,A 8.8135,B 5.6107,C 0.2411,E1 5.7747,E2 443.8085} C_DIS
LIN {X 138.0881,Y 12.9751,Z 179,A 7.3731,B 5.6108,C 0.2385,E1 5.7751,E2 445.1839} C_DIS
LIN {X 138.4041,Y 9.009,Z 179,A 5.8752,B 5.6108,C 0.2409,E1 5.7754,E2 446.6645} C_DIS
LIN {X 138.5936,Y 5.3342,Z 179,A 4.3869,B 5.6106,C 0.2448,E1 5.7756,E2 448.1498} C_DIS
LIN {X 138.6843,Y 1.872,Z 179,A 2.9356,B 5.6104,C 0.2492,E1 5.7756,E2 449.6049} C_DIS
LIN {X 138.6799,Y -2.1333,Z 179,A 1.3277,B 5.6102,C 0.2532,E1 5.7756,E2 451.208} C_DIS
LIN {X 138.5706,Y -5.923,Z 179,A -0.1579,B 5.61,C 0.2564,E1 5.7755,E2 452.6846} C_DIS
LIN {X 138.3629,Y -9.621,Z 179,A -1.5906,B 5.61,C 0.2592,E1 5.7753,E2 454.106} C_DIS
LIN {X 138.08,Y -13.06,Z 179,A -3.1794,B 5.6096,C 0.2658,E1 5.7749,E2 455.7169} C_DIS
LIN {X 137.5756,Y -17.5987,Z 179,A -4.7458,B 5.6096,C 0.2662,E1 5.7744,E2 457.2438} C_DIS
LIN {X 137.014,Y -21.537,Z 179,A -6.4551,B 5.6093,C 0.2719,E1 5.7737,E2 458.9629} C_DIS
LIN {X 136.3264,Y -25.533,Z 179,A -8.0961,B 5.6091,C 0.276,E1 5.7729,E2 460.601} C_DIS
LIN {X 135.6546,Y -28.8883,Z 179,A -9.5384,B 5.6089,C 0.2805,E1 5.7721,E2 462.0481} C_DIS
LIN {X 134.8563,Y -32.4087,Z 179,A -10.977,B 5.6087,C 0.2838,E1 5.7711,E2 463.4812} C_DIS
LIN {X 134.0002,Y -35.7838,Z 179,A -12.2333,B 5.6087,C 0.2849,E1 5.7703,E2 464.7153} C_DIS
LIN {X 133.0688,Y -39.1054,Z 179,A -13.9105,B 5.6083,C 0.2928,E1 5.769,E2 466.4262} C_DIS
LIN {X 131.7173,Y -43.4421,Z 179,A -15.5633,B 5.6082,C 0.2945,E1 5.7676,E2 468.0519} C_DIS
LIN {X 130.5703,Y -46.776,Z 179,A -16.8361,B 5.6082,C 0.2956,E1 5.7664,E2 469.3022} C_DIS
LIN {X 129.3911,Y -49.9454,Z 179,A -18.4081,B 5.6078,C 0.3021,E1 5.7649,E2 470.8981} C_DIS
LIN {X 128.081,Y -53.2147,Z 179,A -19.7687,B 5.6076,C 0.3045,E1 5.7634,E2 472.2478} C_DIS
LIN {X 126.7287,Y -56.3596,Z 179,A -21.1966,B 5.6074,C 0.3084,E1 5.7618,E2 473.6787} C_DIS
LIN {X 125.29,Y -59.4895,Z 179,A -22.5377,B 5.6073,C 0.3109,E1 5.7603,E2 475.0104} C_DIS
LIN {X 123.9904,Y -62.1576,Z 179,A -23.8875,B 5.607,C 0.316,E1 5.7586,E2 476.3775} C_DIS
LIN {X 121.9577,Y -66.0571,Z 179,A -25.6711,B 5.6068,C 0.3201,E1 5.7562,E2 478.1585} C_DIS
LIN {X 119.7172,Y -70.035,Z 179,A -27.5057,B 5.6065,C 0.3241,E1 5.7537,E2 479.9881} C_DIS
LIN {X 116.8876,Y -74.6616,Z 179,A -29.6763,B 5.6063,C 0.3285,E1 5.7505,E2 482.1517} C_DIS
LIN {X 114.5238,Y -78.2395,Z 179,A -31.4063,B 5.6061,C 0.3322,E1 5.7478,E2 483.8779} C_DIS
LIN {X 111.9654,Y -81.859,Z 179,A -33.0567,B 5.606,C 0.3338,E1 5.7452,E2 485.5065} C_DIS
LIN {X 110.3922,Y -83.9686,Z 179,A -34.3318,B 5.6057,C 0.3391,E1 5.743,E2 486.807} C_DIS
LIN {X 107.239,Y -87.9596,Z 179,A -36.2528,B 5.6055,C 0.3412,E1 5.7397,E2 488.7065} C_DIS
LIN {X 103.5057,Y -92.3238,Z 179,A -38.668,B 5.6052,C 0.3471,E1 5.7352,E2 491.1294} C_DIS
LIN {X 98.8779,Y -97.2637,Z 179,A -41.381,B 5.6049,C 0.3518,E1 5.73,E2 493.8339} C_DIS
LIN {X 95.5855,Y -100.5015,Z 179,A -43.2706,B 5.6046,C 0.3555,E1 5.7262,E2 495.723} C_DIS
LIN {X 92.5172,Y -103.3325,Z 179,A -45.3894,B 5.6041,C 0.3648,E1 5.7217,E2 497.8944} C_DIS
LIN {X 89.0119,Y -106.3668,Z 179,A -46.8161,B 5.6043,C 0.3612,E1 5.7188,E2 499.2593} C_DIS
LIN {X 86.7864,Y -108.191,Z 179,A -48.1279,B 5.604,C 0.3653,E1 5.7159,E2 500.5882} C_DIS
LIN {X 82.7749,Y -111.2895,Z 179,A -49.9414,B 5.604,C 0.3649,E1 5.712,E2 502.3669} C_DIS
LIN {X 78.0592,Y -114.647,Z 179,A -52.4506,B 5.6037,C 0.3708,E1 5.7062,E2 504.8935} C_DIS
LIN {X 74.4493,Y -117.0235,Z 179,A -54.1551,B 5.6035,C 0.3726,E1 5.7022,E2 506.5888} C_DIS
LIN {X 71.558,Y -118.8131,Z 179,A -55.6163,B 5.6033,C 0.3756,E1 5.6987,E2 508.0585} C_DIS
LIN {X 66.7519,Y -121.5787,Z 179,A -57.8482,B 5.6032,C 0.3782,E1 5.6933,E2 510.2847} C_DIS
LIN {X 63.1909,Y -123.4644,Z 179,A -59.4171,B 5.6031,C 0.3792,E1 5.6894,E2 511.8422} C_DIS
LIN {X 59.7908,Y -125.1461,Z 179,A -60.8884,B 5.6031,C 0.3799,E1 5.6858,E2 513.3022} C_DIS
LIN {X 56.7612,Y -126.5491,Z 179,A -62.2609,B 5.6029,C 0.3816,E1 5.6823,E2 514.6748} C_DIS
LIN {X 53.7412,Y -127.8612,Z 179,A -63.6554,B 5.6028,C 0.3838,E1 5.6787,E2 516.0749} C_DIS
LIN {X 50.6305,Y -129.1248,Z 179,A -64.9654,B 5.6028,C 0.3843,E1 5.6753,E2 517.3758} C_DIS
LIN {X 47.9205,Y -130.1566,Z 179,A -66.3675,B 5.6025,C 0.3885,E1 5.6716,E2 518.8056} C_DIS
LIN {X 44.0376,Y -131.519,Z 179,A -67.8869,B 5.6025,C 0.3877,E1 5.6676,E2 520.3025} C_DIS
LIN {X 40.886,Y -132.5328,Z 179,A -69.1198,B 5.6025,C 0.3872,E1 5.6644,E2 521.5185} C_DIS
LIN {X 37.3118,Y -133.5828,Z 179,A -70.6367,B 5.6025,C 0.3883,E1 5.6603,E2 523.0337} C_DIS
LIN {X 33.8634,Y -134.4986,Z 179,A -72.5342,B 5.602,C 0.3953,E1 5.655,E2 524.9876} C_DIS
LIN {X 30.4967,Y -135.3021,Z 179,A -73.7501,B 5.6021,C 0.3935,E1 5.6518,E2 526.1764} C_DIS
LIN {X 26.6142,Y -136.1198,Z 179,A -75.3553,B 5.6021,C 0.3942,E1 5.6474,E2 527.7782} C_DIS
LIN {X 22.6278,Y -136.8378,Z 179,A -77.5871,B 5.6015,C 0.4026,E1 5.641,E2 530.0837} C_DIS
LIN {X 17.2907,Y -137.616,Z 179,A -79.2859,B 5.6019,C 0.3967,E1 5.6365,E2 531.7151} C_DIS
LIN {X 13.2599,Y -138.0608,Z 179,A -80.8171,B 5.6019,C 0.3955,E1 5.6323,E2 533.2282} C_DIS
LIN {X 9.6777,Y -138.3587,Z 179,A -82.2925,B 5.6019,C 0.3959,E1 5.6282,E2 534.7032} C_DIS
LIN {X 5.7328,Y -138.578,Z 179,A -83.9008,B 5.6019,C 0.396,E1 5.6237,E2 536.3091} C_DIS
LIN {X 1.9679,Y -138.6827,Z 179,A -85.6017,B 5.6018,C 0.3982,E1 5.6189,E2 538.0298} C_DIS
LIN {X 1.9679,Y -138.6827,Z 179,A -85.6017,B 5.6018,C 0.3982,E1 5.6189,E2 538.0298} C_DIS
Enddeposition()
LIN {X 0.9952,Y -139.5939,Z 179,A -85.3564,B 5.568,C 0.3925,E1 5.5856,E2 537.7415} C_DIS
Startdeposition()
$VEL.CP = VEL_PRINT
LIN {X 4.6173,Y -139.5251,Z 179,A -83.6257,B 5.5682,C 0.3891,E1 5.5905,E2 535.9777} C_DIS
LIN {X 8.5534,Y -139.3372,Z 179,A -82.1482,B 5.5682,C 0.3904,E1 5.5946,E2 534.518} C_DIS
LIN {X 11.9723,Y -139.0853,Z 179,A -80.7125,B 5.5682,C 0.3896,E1 5.5986,E2 533.0778} C_DIS
LIN {X 15.5933,Y -138.7274,Z 179,A -79.2502,B 5.5682,C 0.3894,E1 5.6027,E2 531.6188} C_DIS
LIN {X 19.4991,Y -138.2311,Z 179,A -77.1805,B 5.5687,C 0.3824,E1 5.6086,E2 529.4874} C_DIS
LIN {X 23.7411,Y -137.5679,Z 179,A -75.8843,B 5.5683,C 0.3877,E1 5.612,E2 528.2527} C_DIS
LIN {X 29.0485,Y -136.5442,Z 179,A -73.8215,B 5.5683,C 0.3883,E1 5.6176,E2 526.2092} C_DIS
LIN {X 35.0378,Y -135.1325,Z 179,A -71.0544,B 5.5687,C 0.383,E1 5.6252,E2 523.4085} C_DIS
LIN {X 39.8613,Y -133.7888,Z 179,A -69.1448,B 5.5687,C 0.3832,E1 5.6303,E2 521.517} C_DIS
LIN {X 42.6686,Y -132.9185,Z 179,A -67.927,B 5.5687,C 0.3819,E1 5.6335,E2 520.2967} C_DIS
LIN {X 46.2769,Y -131.7068,Z 179,A -66.4118,B 5.5688,C 0.3809,E1 5.6375,E2 518.7868} C_DIS
LIN {X 49.008,Y -130.7139,Z 179,A -65.1335,B 5.569,C 0.3784,E1 5.6409,E2 517.4962} C_DIS
LIN {X 52.7255,Y -129.2603,Z 179,A -63.5663,B 5.569,C 0.3775,E1 5.6449,E2 515.9373} C_DIS
LIN {X 55.8947,Y -127.9217,Z 179,A -62.2042,B 5.5691,C 0.3764,E1 5.6484,E2 514.5808} C_DIS
LIN {X 58.7436,Y -126.6376,Z 179,A -60.8741,B 5.5693,C 0.3741,E1 5.6518,E2 513.2433} C_DIS
LIN {X 62.3352,Y -124.9104,Z 179,A -59.2819,B 5.5693,C 0.3725,E1 5.6558,E2 511.6558} C_DIS
LIN {X 65.2336,Y -123.4204,Z 179,A -57.9328,B 5.5695,C 0.3704,E1 5.6591,E2 510.304} C_DIS
LIN {X 71.6372,Y -119.819,Z 179,A -55.131,B 5.5696,C 0.369,E1 5.6659,E2 507.5285} C_DIS
LIN {X 75.6118,Y -117.3518,Z 179,A -52.9871,B 5.57,C 0.3626,E1 5.671,E2 505.3532} C_DIS
LIN {X 80.0912,Y -114.341,Z 179,A -50.7301,B 5.5703,C 0.3582,E1 5.6762,E2 503.0889} C_DIS
LIN {X 83.5045,Y -111.8725,Z 179,A -49.0672,B 5.5704,C 0.3561,E1 5.6799,E2 501.4333} C_DIS
LIN {X 87.3526,Y -108.8948,Z 179,A -47.13,B 5.5706,C 0.3533,E1 5.6842,E2 499.5024} C_DIS
LIN {X 91.6385,Y -105.3129,Z 179,A -45.0628,B 5.5706,C 0.3523,E1 5.6885,E2 497.4633} C_DIS
LIN {X 94.4213,Y -102.8254,Z 179,A -43.4106,B 5.571,C 0.3474,E1 5.692,E2 495.7937} C_DIS
LIN {X 97.7207,Y -99.695,Z 179,A -41.5742,B 5.5712,C 0.3441,E1 5.6957,E2 493.9597} C_DIS
LIN {X 100.9874,Y -96.3845,Z 179,A -39.8153,B 5.5712,C 0.3423,E1 5.699,E2 492.219} C_DIS
LIN {X 103.8168,Y -93.3304,Z 179,A -38.2432,B 5.5714,C 0.3407,E1 5.702,E2 490.6636} C_DIS
LIN {X 105.9948,Y -90.8496,Z 179,A -36.7776,B 5.5717,C 0.336,E1 5.7047,E2 489.1821} C_DIS
LIN {X 108.5152,Y -87.8234,Z 179,A -34.4161,B 5.5726,C 0.3208,E1 5.709,E2 486.7196} C_DIS
LIN {X 112.3001,Y -82.9291,Z 179,A -32.7344,B 5.5721,C 0.3282,E1 5.7117,E2 485.1502} C_DIS
LIN {X 114.4826,Y -79.8887,Z 179,A -31.1115,B 5.5724,C 0.3232,E1 5.7143,E2 483.5145} C_DIS
LIN {X 117.0573,Y -76.066,Z 179,A -28.9455,B 5.5729,C 0.3143,E1 5.7177,E2 481.3102} C_DIS
LIN {X 119.2518,Y -72.5783,Z 179,A -27.6047,B 5.5729,C 0.3156,E1 5.7196,E2 480.0146} C_DIS
LIN {X 121.5459,Y -68.6668,Z 179,A -25.7696,B 5.5731,C 0.3113,E1 5.7221,E2 478.1812} C_DIS
LIN {X 123.6227,Y -64.8482,Z 179,A -24.1329,B 5.5732,C 0.3091,E1 5.7242,E2 476.5623} C_DIS
LIN {X 125.3334,Y -61.4776,Z 179,A -22.5978,B 5.5734,C 0.3053,E1 5.7262,E2 475.0279} C_DIS
LIN {X 126.8555,Y -58.2723,Z 179,A -21.1931,B 5.5736,C 0.3023,E1 5.7278,E2 473.6288} C_DIS
LIN {X 128.4445,Y -54.6855,Z 179,A -19.6381,B 5.5738,C 0.2989,E1 5.7295,E2 472.0797} C_DIS
LIN {X 129.6129,Y -51.8508,Z 179,A -18.3963,B 5.574,C 0.2958,E1 5.7308,E2 470.8388} C_DIS
LIN {X 130.7942,Y -48.7935,Z 179,A -17.0862,B 5.5741,C 0.2927,E1 5.7321,E2 469.5322} C_DIS
LIN {X 131.92,Y -45.662,Z 179,A -15.7186,B 5.5743,C 0.289,E1 5.7334,E2 468.1631} C_DIS
LIN {X 133.1089,Y -42.0729,Z 179,A -13.6469,B 5.5749,C 0.2765,E1 5.7352,E2 466.0214} C_DIS
LIN {X 134.5627,Y -37.1621,Z 179,A -12.2353,B 5.5747,C 0.2817,E1 5.7362,E2 464.6992} C_DIS
LIN {X 135.5872,Y -33.2317,Z 179,A -10.6844,B 5.5748,C 0.2789,E1 5.7373,E2 463.1621} C_DIS
LIN {X 136.6367,Y -28.6182,Z 179,A -8.4975,B 5.5753,C 0.2696,E1 5.7386,E2 460.9415} C_DIS
LIN {X 137.5162,Y -24.0326,Z 179,A -6.826,B 5.5753,C 0.268,E1 5.7394,E2 459.3005} C_DIS
LIN {X 138.0145,Y -20.9787,Z 179,A -5.5289,B 5.5755,C 0.264,E1 5.74,E2 457.9988} C_DIS
LIN {X 138.5825,Y -16.8213,Z 179,A -3.8265,B 5.5758,C 0.2594,E1 5.7406,E2 456.2975} C_DIS
LIN {X 138.9633,Y -13.3117,Z 179,A -2.4843,B 5.5758,C 0.257,E1 5.741,E2 454.9681} C_DIS
LIN {X 139.2873,Y -9.3633,Z 179,A -0.7729,B 5.5761,C 0.251,E1 5.7413,E2 453.2443} C_DIS
LIN {X 139.4947,Y -5.4092,Z 179,A 0.7041,B 5.5762,C 0.2487,E1 5.7415,E2 451.7854} C_DIS
LIN {X 139.5958,Y -1.1507,Z 179,A 2.4347,B 5.5765,C 0.244,E1 5.7415,E2 450.0557} C_DIS
LIN {X 139.5742,Y 2.6827,Z 179,A 4.0473,B 5.5767,C 0.2389,E1 5.7415,E2 448.4367} C_DIS
LIN {X 139.4216,Y 7.0455,Z 179,A 5.6666,B 5.5767,C 0.2365,E1 5.7413,E2 446.8385} C_DIS
LIN {X 139.2172,Y 10.3247,Z 179,A 7.0265,B 5.5769,C 0.2325,E1 5.7411,E2 445.4763} C_DIS
LIN {X 138.8876,Y 14.1,Z 179,A 8.4876,B 5.5771,C 0.2296,E1 5.7407,E2 444.0263} C_DIS
LIN {X 138.3623,Y 18.5474,Z 179,A 10.9654,B 5.5777,C 0.2143,E1 5.7398,E2 441.4636} C_DIS
LIN {X 137.5212,Y 24.005,Z 179,A 12.4173,B 5.5774,C 0.2208,E1 5.7391,E2 440.1165} C_DIS
LIN {X 136.9379,Y 27.1381,Z 179,A 13.9946,B 5.5777,C 0.2129,E1 5.7383,E2 438.5033} C_DIS
LIN {X 135.9831,Y 31.5717,Z 179,A 15.5634,B 5.5777,C 0.2123,E1 5.7373,E2 436.9713} C_DIS
LIN {X 135.2699,Y 34.4967,Z 179,A 16.8131,B 5.5779,C 0.2087,E1 5.7365,E2 435.719} C_DIS
LIN {X 134.4087,Y 37.7127,Z 179,A 18.1589,B 5.578,C 0.2053,E1 5.7355,E2 434.3751} C_DIS
LIN {X 133.3061,Y 41.4462,Z 179,A 19.6762,B 5.5781,C 0.2022,E1 5.7343,E2 432.8672} C_DIS
LIN {X 132.3311,Y 44.4581,Z 179,A 20.9884,B 5.5783,C 0.1984,E1 5.7331,E2 431.5525} C_DIS
LIN {X 130.9343,Y 48.4196,Z 179,A 22.9244,B 5.5785,C 0.1905,E1 5.7313,E2 429.5882} C_DIS
LIN {X 129.7743,Y 51.447,Z 179,A 24.4037,B 5.5787,C 0.1847,E1 5.7297,E2 428.0888} C_DIS
LIN {X 128.1589,Y 55.3461,Z 179,A 25.3583,B 5.5785,C 0.1922,E1 5.7288,E2 427.2337} C_DIS
LIN {X 126.6114,Y 58.8003,Z 179,A 27.2855,B 5.5788,C 0.1824,E1 5.7265,E2 425.2577} C_DIS
LIN {X 125.0463,Y 62.0597,Z 179,A 28.6234,B 5.5788,C 0.1809,E1 5.7249,E2 423.9379} C_DIS
LIN {X 123.4195,Y 65.2352,Z 179,A 30.0583,B 5.579,C 0.1776,E1 5.723,E2 422.5061} C_DIS
LIN {X 120.9688,Y 69.6763,Z 179,A 32.5036,B 5.5793,C 0.1669,E1 5.7196,E2 420.013} C_DIS
LIN {X 118.8203,Y 73.2823,Z 179,A 33.6529,B 5.5791,C 0.1714,E1 5.718,E2 418.9369} C_DIS
LIN {X 117.0088,Y 76.1407,Z 179,A 35.1942,B 5.5793,C 0.1658,E1 5.7157,E2 417.3755} C_DIS
LIN {X 114.7642,Y 79.484,Z 179,A 36.819,B 5.5794,C 0.1623,E1 5.7131,E2 415.7537} C_DIS
LIN {X 112.1941,Y 83.0726,Z 179,A 38.6138,B 5.5795,C 0.1584,E1 5.7102,E2 413.9605} C_DIS
LIN {X 109.4917,Y 86.6035,Z 179,A 40.7054,B 5.5798,C 0.1503,E1 5.7065,E2 411.8339} C_DIS
LIN {X 107.0044,Y 89.6576,Z 179,A 41.881,B 5.5797,C 0.1533,E1 5.7045,E2 410.7144} C_DIS
LIN {X 104.4718,Y 92.5964,Z 179,A 43.5497,B 5.5797,C 0.1488,E1 5.7014,E2 409.0355} C_DIS
LIN {X 101.4551,Y 95.8922,Z 179,A 45.3044,B 5.5799,C 0.1461,E1 5.6981,E2 407.2905} C_DIS
LIN {X 98.3849,Y 99.0396,Z 179,A 47.629,B 5.5802,C 0.1348,E1 5.6934,E2 404.8987} C_DIS
LIN {X 94.6689,Y 102.5978,Z 179,A 49.0522,B 5.58,C 0.1407,E1 5.6906,E2 403.5634} C_DIS
LIN {X 91.4138,Y 105.5089,Z 179,A 50.9653,B 5.5801,C 0.1356,E1 5.6866,E2 401.6347} C_DIS
LIN {X 87.9522,Y 108.4112,Z 179,A 52.8137,B 5.5802,C 0.1323,E1 5.6826,E2 399.7867} C_DIS
LIN {X 84.3102,Y 111.2668,Z 179,A 54.6627,B 5.5802,C 0.1297,E1 5.6785,E2 397.9439} C_DIS
LIN {X 80.3126,Y 114.1848,Z 179,A 56.8589,B 5.5804,C 0.1239,E1 5.6735,E2 395.7265} C_DIS
LIN {X 77.436,Y 116.1555,Z 179,A 57.9346,B 5.5804,C 0.1267,E1 5.6711,E2 394.6959} C_DIS
LIN {X 74.1937,Y 118.2534,Z 179,A 59.6396,B 5.5804,C 0.1225,E1 5.6671,E2 392.9757} C_DIS
LIN {X 70.3905,Y 120.556,Z 179,A 61.4494,B 5.5804,C 0.12,E1 5.6627,E2 391.1678} C_DIS
LIN {X 66.3486,Y 122.8267,Z 179,A 63.436,B 5.5806,C 0.1162,E1 5.6578,E2 389.1706} C_DIS
LIN {X 61.7049,Y 125.2213,Z 179,A 65.6716,B 5.5806,C 0.1121,E1 5.6522,E2 386.9235} C_DIS
LIN {X 58.3883,Y 126.8019,Z 179,A 66.7763,B 5.5806,C 0.1158,E1 5.6495,E2 385.87} C_DIS
LIN {X 55.3983,Y 128.1363,Z 179,A 68.187,B 5.5806,C 0.1133,E1 5.6459,E2 384.451} C_DIS
LIN {X 51.9004,Y 129.593,Z 179,A 69.7151,B 5.5806,C 0.112,E1 5.642,E2 382.9265} C_DIS
LIN {X 48.5809,Y 130.8738,Z 179,A 71.1499,B 5.5806,C 0.1108,E1 5.6382,E2 381.4952} C_DIS
LIN {X 44.3578,Y 132.3645,Z 179,A 73.0491,B 5.5807,C 0.1082,E1 5.6332,E2 379.5886} C_DIS
LIN {X 40.5314,Y 133.5861,Z 179,A 74.5752,B 5.5807,C 0.1084,E1 5.6292,E2 378.0783} C_DIS
LIN {X 37.0181,Y 134.6029,Z 179,A 76.0785,B 5.5807,C 0.1072,E1 5.6251,E2 376.575} C_DIS
LIN {X 31.739,Y 135.9449,Z 179,A 78.3866,B 5.5807,C 0.1046,E1 5.6188,E2 374.2584} C_DIS
LIN {X 26.9334,Y 136.9784,Z 179,A 80.2596,B 5.5807,C 0.1053,E1 5.6138,E2 372.4042} C_DIS
LIN {X 23.4427,Y 137.6177,Z 179,A 82.1341,B 5.5809,C 0.0991,E1 5.6085,E2 370.4774} C_DIS
LIN {X 19.7336,Y 138.1975,Z 179,A 83.493,B 5.5809,C 0.1008,E1 5.6048,E2 369.1419} C_DIS
LIN {X 15.1163,Y 138.7787,Z 179,A 85.2278,B 5.5809,C 0.1023,E1 5.6,E2 367.4299} C_DIS
LIN {X 11.5913,Y 139.1175,Z 179,A 86.6788,B 5.5809,C 0.1019,E1 5.596,E2 365.9798} C_DIS
LIN {X 7.4104,Y 139.4033,Z 179,A 88.3991,B 5.5809,C 0.1016,E1 5.5912,E2 364.2601} C_DIS
LIN {X 3.7325,Y 139.5497,Z 179,A 89.8631,B 5.5809,C 0.1019,E1 5.5871,E2 362.8026} C_DIS
LIN {X 0.3099,Y 139.6,Z 179,A 91.2572,B 5.5809,C 0.1019,E1 5.5832,E2 361.4105} C_DIS
LIN {X -3.6984,Y 139.5506,Z 179,A 92.9279,B 5.5809,C 0.1017,E1 5.5786,E2 359.7374} C_DIS
LIN {X -7.7429,Y 139.3865,Z 179,A 94.5524,B 5.5809,C 0.1023,E1 5.574,E2 358.1183} C_DIS
LIN {X -12.7215,Y 139.02,Z 179,A 96.791,B 5.5809,C 0.1004,E1 5.5677,E2 355.8569} C_DIS
LIN {X -17.0403,Y 138.5564,Z 179,A 98.4952,B 5.5809,C 0.1019,E1 5.563,E2 354.1635} C_DIS
LIN {X -25.501,Y 137.2523,Z 179,A 102.0968,B 5.5809,C 0.1024,E1 5.5531,E2 350.5529} C_DIS
LIN {X -29.3564,Y 136.4777,Z 179,A 103.6174,B 5.5809,C 0.1043,E1 5.549,E2 349.045} C_DIS
LIN {X -32.9989,Y 135.6433,Z 179,A 105.1076,B 5.5808,C 0.1058,E1 5.5449,E2 347.5611} C_DIS
LIN {X -38.2671,Y 134.2536,Z 179,A 107.329,B 5.5808,C 0.1075,E1 5.539,E2 345.3431} C_DIS
LIN {X -41.2184,Y 133.3758,Z 179,A 108.6039,B 5.5808,C 0.1084,E1 5.5355,E2 344.0676} C_DIS
LIN {X -44.3673,Y 132.3614,Z 179,A 110.0052,B 5.5808,C 0.1091,E1 5.5318,E2 342.6617} C_DIS
LIN {X -47.6429,Y 131.218,Z 179,A 111.4987,B 5.5808,C 0.1096,E1 5.5279,E2 341.1604} C_DIS
LIN {X -53.0862,Y 129.1136,Z 179,A 114.1435,B 5.5808,C 0.1093,E1 5.5209,E2 338.4859} C_DIS
LIN {X -56.0736,Y 127.8443,Z 179,A 115.2118,B 5.5806,C 0.1137,E1 5.5183,E2 337.4518} C_DIS
LIN {X -60.0816,Y 126.0083,Z 179,A 117.103,B 5.5806,C 0.1149,E1 5.5135,E2 335.5515} C_DIS
LIN {X -63.6095,Y 124.265,Z 179,A 118.6962,B 5.5806,C 0.1172,E1 5.5095,E2 333.9623} C_DIS
LIN {X -67.1906,Y 122.3684,Z 179,A 120.4285,B 5.5806,C 0.1187,E1 5.5052,E2 332.2226} C_DIS
LIN {X -71.1425,Y 120.1138,Z 179,A 122.3588,B 5.5805,C 0.1206,E1 5.5005,E2 330.2858} C_DIS
LIN {X -74.9927,Y 117.7482,Z 179,A 124.2468,B 5.5805,C 0.123,E1 5.4961,E2 328.395} C_DIS
LIN {X -78.729,Y 115.2835,Z 179,A 126.1064,B 5.5804,C 0.1257,E1 5.4918,E2 326.5341} C_DIS
LIN {X -84.1969,Y 111.3522,Z 179,A 129.04,B 5.5803,C 0.1285,E1 5.4851,E2 323.5813} C_DIS
LIN {X -88.7405,Y 107.7669,Z 179,A 131.3446,B 5.5802,C 0.1335,E1 5.4801,E2 321.2876} C_DIS
LIN {X -94.0549,Y 103.1611,Z 179,A 134.7585,B 5.5802,C 0.1335,E1 5.4729,E2 317.8092} C_DIS
LIN {X -97.6884,Y 99.7267,Z 179,A 136.2092,B 5.5799,C 0.1437,E1 5.4701,E2 316.4366} C_DIS
LIN {X -100.5121,Y 96.8806,Z 179,A 138.4758,B 5.58,C 0.1407,E1 5.4656,E2 314.0926} C_DIS
LIN {X -103.7543,Y 93.4002,Z 179,A 140.2088,B 5.5798,C 0.147,E1 5.4624,E2 312.3892} C_DIS
LIN {X -105.9683,Y 90.8804,Z 179,A 141.3374,B 5.5797,C 0.1525,E1 5.4604,E2 311.2933} C_DIS
LIN {X -108.6065,Y 87.7101,Z 179,A 143.1343,B 5.5797,C 0.1552,E1 5.4572,E2 309.4846} C_DIS
LIN {X -112.2132,Y 83.0469,Z 179,A 145.428,B 5.5794,C 0.1619,E1 5.4533,E2 307.2091} C_DIS
LIN {X -114.2818,Y 80.1762,Z 179,A 147.0862,B 5.5794,C 0.1632,E1 5.4506,E2 305.5261} C_DIS
LIN {X -116.8418,Y 76.3978,Z 179,A 148.9924,B 5.5793,C 0.1674,E1 5.4476,E2 303.6173} C_DIS
LIN {X -119.1401,Y 72.7609,Z 179,A 150.8106,B 5.5792,C 0.1711,E1 5.445,E2 301.794} C_DIS
LIN {X -121.4707,Y 68.8003,Z 179,A 152.7512,B 5.579,C 0.1753,E1 5.4422,E2 299.8482} C_DIS
LIN {X -124.1298,Y 63.8752,Z 179,A 155.2481,B 5.579,C 0.1791,E1 5.439,E2 297.3278} C_DIS
LIN {X -126.2544,Y 59.5665,Z 179,A 157.0059,B 5.5787,C 0.1863,E1 5.4369,E2 295.5991} C_DIS
LIN {X -127.6955,Y 56.4105,Z 179,A 158.4733,B 5.5786,C 0.1895,E1 5.4352,E2 294.1273} C_DIS
LIN {X -129.6957,Y 51.6436,Z 179,A 160.7204,B 5.5784,C 0.194,E1 5.4328,E2 291.8662} C_DIS
LIN {X -130.8718,Y 48.5864,Z 179,A 162.1021,B 5.5784,C 0.1972,E1 5.4314,E2 290.4808} C_DIS
LIN {X -132.4013,Y 44.2475,Z 179,A 164.0247,B 5.5781,C 0.202,E1 5.4297,E2 288.5554} C_DIS
LIN {X -133.6614,Y 40.2851,Z 179,A 165.6596,B 5.5779,C 0.2073,E1 5.4283,E2 286.9312} C_DIS
LIN {X -134.4645,Y 37.513,Z 179,A 166.9342,B 5.5779,C 0.2097,E1 5.4273,E2 285.6462} C_DIS
LIN {X -135.4263,Y 33.8804,Z 179,A 168.4794,B 5.5777,C 0.2139,E1 5.4263,E2 284.1019} C_DIS
LIN {X -136.1943,Y 30.6475,Z 179,A 169.8869,B 5.5776,C 0.2173,E1 5.4254,E2 282.6899} C_DIS
LIN {X -137.2147,Y 25.6975,Z 179,A 172.2487,B 5.5774,C 0.2204,E1 5.4241,E2 280.293} C_DIS
LIN {X -137.9578,Y 21.3455,Z 179,A 173.8585,B 5.5772,C 0.2274,E1 5.4234,E2 278.7108} C_DIS
LIN {X -138.4204,Y 18.1044,Z 179,A 175.2734,B 5.577,C 0.2306,E1 5.4228,E2 277.2878} C_DIS
LIN {X -139.1187,Y 11.577,Z 179,A 178.0771,B 5.5767,C 0.2372,E1 5.4221,E2 274.4724} C_DIS
LIN {X -139.4755,Y 5.9019,Z 179,A -179.7135,B 5.5764,C 0.245,E1 5.4217,E2 272.2809} C_DIS
LIN {X -139.5773,Y 2.4991,Z 179,A -177.4643,B 5.5766,C 0.241,E1 5.4216,E2 269.9226} C_DIS
LIN {X -139.572,Y -2.8193,Z 179,A -175.3175,B 5.5763,C 0.2475,E1 5.4216,E2 267.7822} C_DIS
LIN {X -139.3933,Y -7.6091,Z 179,A -173.9105,B 5.5758,C 0.2584,E1 5.4219,E2 266.4493} C_DIS
LIN {X -139.1558,Y -11.138,Z 179,A -171.8379,B 5.5758,C 0.2567,E1 5.4224,E2 264.2972} C_DIS
LIN {X -138.708,Y -15.7697,Z 179,A -170.1867,B 5.5755,C 0.2645,E1 5.4229,E2 262.6811} C_DIS
LIN {X -138.1961,Y -19.7439,Z 179,A -168.6743,B 5.5752,C 0.2704,E1 5.4234,E2 261.1869} C_DIS
LIN {X -137.6613,Y -23.1816,Z 179,A -167.2669,B 5.575,C 0.2746,E1 5.424,E2 259.7832} C_DIS
LIN {X -136.9622,Y -27.0181,Z 179,A -165.4434,B 5.575,C 0.277,E1 5.425,E2 257.9319} C_DIS
LIN {X -136.0597,Y -31.2365,Z 179,A -163.8297,B 5.5746,C 0.2834,E1 5.426,E2 256.3397} C_DIS
LIN {X -135.2427,Y -34.6039,Z 179,A -162.38,B 5.5744,C 0.287,E1 5.427,E2 254.8873} C_DIS
LIN {X -134.3372,Y -37.9681,Z 179,A -160.8687,B 5.5743,C 0.2901,E1 5.4281,E2 253.3663} C_DIS
LIN {X -133.2848,Y -41.5157,Z 179,A -159.2781,B 5.5741,C 0.2935,E1 5.4294,E2 251.7673} C_DIS
LIN {X -132.0506,Y -45.2853,Z 179,A -157.362,B 5.574,C 0.2951,E1 5.4311,E2 249.8145} C_DIS
LIN {X -130.9398,Y -48.4043,Z 179,A -156.0241,B 5.5738,C 0.2989,E1 5.4324,E2 248.4802} C_DIS
LIN {X -129.3252,Y -52.5647,Z 179,A -154.3623,B 5.5734,C 0.3054,E1 5.4341,E2 246.8415} C_DIS
LIN {X -127.7844,Y -56.2118,Z 179,A -152.4542,B 5.5734,C 0.3068,E1 5.4363,E2 244.8974} C_DIS
LIN {X -125.7392,Y -60.6448,Z 179,A -150.6706,B 5.573,C 0.314,E1 5.4384,E2 243.1435} C_DIS
LIN {X -124.2386,Y -63.6614,Z 179,A -149.2204,B 5.5728,C 0.3168,E1 5.4402,E2 241.6851} C_DIS
LIN {X -120.1818,Y -71.0275,Z 179,A -145.8212,B 5.5723,C 0.3258,E1 5.4448,E2 238.2947} C_DIS
LIN {X -118.4014,Y -73.9568,Z 179,A -144.0937,B 5.5723,C 0.3259,E1 5.4474,E2 236.5257} C_DIS
LIN {X -116.1048,Y -77.512,Z 179,A -142.4132,B 5.572,C 0.3306,E1 5.45,E2 234.8533} C_DIS
LIN {X -113.4958,Y -81.2844,Z 179,A -140.5061,B 5.5718,C 0.3346,E1 5.4531,E2 232.9437} C_DIS
LIN {X -111.138,Y -84.4804,Z 179,A -139.0882,B 5.5714,C 0.3404,E1 5.4554,E2 231.5542} C_DIS
LIN {X -109.2602,Y -86.8944,Z 179,A -137.5446,B 5.5714,C 0.3402,E1 5.4581,E2 229.9731} C_DIS
LIN {X -106.3534,Y -90.4289,Z 179,A -135.6295,B 5.5712,C 0.3438,E1 5.4616,E2 228.0538} C_DIS
LIN {X -103.4612,Y -93.7242,Z 179,A -133.7888,B 5.571,C 0.347,E1 5.465,E2 226.2081} C_DIS
LIN {X -100.4668,Y -96.9274,Z 179,A -131.9425,B 5.5708,C 0.3501,E1 5.4686,E2 224.3561} C_DIS
LIN {X -97.3029,Y -100.1032,Z 179,A -130.0583,B 5.5706,C 0.3532,E1 5.4723,E2 222.4665} C_DIS
LIN {X -93.9826,Y -103.2267,Z 179,A -128.1636,B 5.5704,C 0.3564,E1 5.4762,E2 220.5689} C_DIS
LIN {X -90.5005,Y -106.2925,Z 179,A -126.2354,B 5.5702,C 0.3596,E1 5.4803,E2 218.6378} C_DIS
LIN {X -86.848,Y -109.2972,Z 179,A -124.2975,B 5.57,C 0.3629,E1 5.4845,E2 216.7006} C_DIS
LIN {X -81.8299,Y -113.1027,Z 179,A -121.3639,B 5.57,C 0.3632,E1 5.4912,E2 213.721} C_DIS
LIN {X -78.648,Y -115.3391,Z 179,A -120.2383,B 5.5695,C 0.3709,E1 5.4936,E2 212.658} C_DIS
LIN {X -75.815,Y -117.2201,Z 179,A -118.7538,B 5.5695,C 0.372,E1 5.4971,E2 211.1618} C_DIS
LIN {X -72.564,Y -119.2604,Z 179,A -116.9936,B 5.5694,C 0.372,E1 5.5014,E2 209.3771} C_DIS
LIN {X -68.5722,Y -121.5991,Z 179,A -115.0558,B 5.5693,C 0.3741,E1 5.5061,E2 207.434} C_DIS
LIN {X -65.3296,Y -123.3699,Z 179,A -113.0038,B 5.5695,C 0.3698,E1 5.5113,E2 205.3104} C_DIS
LIN {X -60.5748,Y -125.7726,Z 179,A -111.4171,B 5.5689,C 0.3793,E1 5.5151,E2 203.8037} C_DIS
LIN {X -56.8406,Y -127.5031,Z 179,A -109.7242,B 5.5688,C 0.3811,E1 5.5194,E2 202.1101} C_DIS
LIN {X -53.2027,Y -129.065,Z 179,A -108.1083,B 5.5687,C 0.3828,E1 5.5236,E2 200.4953} C_DIS
LIN {X -49.7099,Y -130.451,Z 179,A -105.9665,B 5.5691,C 0.377,E1 5.5294,E2 198.2732} C_DIS
LIN {X -45.0962,Y -132.1162,Z 179,A -104.5576,B 5.5685,C 0.386,E1 5.5329,E2 196.9447} C_DIS
LIN {X -42.3188,Y -133.0303,Z 179,A -103.3522,B 5.5684,C 0.3868,E1 5.5361,E2 195.7382} C_DIS
LIN {X -39.1937,Y -133.9842,Z 179,A -101.9321,B 5.5684,C 0.3868,E1 5.5399,E2 194.3074} C_DIS
LIN {X -34.0858,Y -135.3742,Z 179,A -99.5935,B 5.5684,C 0.3861,E1 5.5463,E2 191.9461} C_DIS
LIN {X -28.9975,Y -136.5552,Z 179,A -97.5973,B 5.5682,C 0.389,E1 5.5517,E2 189.969} C_DIS
LIN {X -24.2022,Y -137.4859,Z 179,A -95.6773,B 5.5682,C 0.3908,E1 5.5569,E2 188.0597} C_DIS
LIN {X -21.0685,Y -138.0006,Z 179,A -94.3306,B 5.5682,C 0.3908,E1 5.5606,E2 186.7068} C_DIS
LIN {X -17.2917,Y -138.5264,Z 179,A -92.6265,B 5.5682,C 0.3893,E1 5.5654,E2 184.9836} C_DIS
LIN {X -13.2622,Y -138.9681,Z 179,A -91.0717,B 5.5682,C 0.391,E1 5.5697,E2 183.4427} C_DIS
LIN {X -9.3751,Y -139.2865,Z 179,A -89.356,B 5.5682,C 0.3897,E1 5.5745,E2 181.7111} C_DIS
LIN {X -5.4504,Y -139.4931,Z 179,A -87.8372,B 5.5682,C 0.3909,E1 5.5787,E2 180.204} C_DIS
LIN {X -1.6487,Y -139.5914,Z 179,A -86.1844,B 5.5682,C 0.3896,E1 5.5834,E2 178.5383} C_DIS
LIN {X 0.9952,Y -139.5939,Z 179,A -85.3543,B 5.568,C 0.3927,E1 5.5856,E2 177.7416} C_DIS
Enddeposition()
LIN {X 0.9952,Y -139.5939,Z 179,A -85.3543,B 5.568,C 0.3927,E1 5.5856,E2 177.7416} C_DIS
Startdeposition()
$VEL.CP = VEL_PRINT
LIN {X -0.8909,Y -140.5001,Z 179,A -86.5486,B 5.4423,C 0.3996,E1 5.457,E2 179.0613} C_DIS
LIN {X -4.701,Y -140.4263,Z 179,A -88.1434,B 5.4423,C 0.4001,E1 5.4525,E2 180.6622} C_DIS
LIN {X -8.4529,Y -140.2484,Z 179,A -89.6224,B 5.4423,C 0.3994,E1 5.4484,E2 182.1349} C_DIS
LIN {X -11.9803,Y -139.9912,Z 179,A -91.0536,B 5.4423,C 0.3992,E1 5.4444,E2 183.5651} C_DIS
LIN {X -16.2768,Y -139.5572,Z 179,A -92.8927,B 5.4423,C 0.3998,E1 5.4393,E2 185.4153} C_DIS
LIN {X -20.2322,Y -139.0388,Z 179,A -94.4552,B 5.4423,C 0.3986,E1 5.435,E2 186.9699} C_DIS
LIN {X -23.4877,Y -138.526,Z 179,A -95.8796,B 5.4423,C 0.3991,E1 5.431,E2 188.4054} C_DIS
LIN {X -27.2307,Y -137.8409,Z 179,A -97.3897,B 5.4423,C 0.398,E1 5.4269,E2 189.9105} C_DIS
LIN {X -30.8949,Y -137.0643,Z 179,A -98.9466,B 5.4424,C 0.3976,E1 5.4226,E2 191.4718} C_DIS
LIN {X -33.9111,Y -136.3505,Z 179,A -100.0803,B 5.4426,C 0.3953,E1 5.4196,E2 192.5885} C_DIS
LIN {X -38.5862,Y -135.1023,Z 179,A -102.1893,B 5.4426,C 0.3957,E1 5.4139,E2 194.7161} C_DIS
LIN {X -42.3754,Y -133.9605,Z 179,A -103.6616,B 5.4428,C 0.3929,E1 5.41,E2 196.1699} C_DIS
LIN {X -47.7345,Y -132.1452,Z 179,A -106.1731,B 5.4428,C 0.3934,E1 5.4033,E2 198.709} C_DIS
LIN {X -52.0526,Y -130.5056,Z 179,A -108.055,B 5.4428,C 0.3916,E1 5.3984,E2 200.591} C_DIS
LIN {X -55.4894,Y -129.081,Z 179,A -109.7186,B 5.4428,C 0.3918,E1 5.3941,E2 202.2741} C_DIS
LIN {X -60.2076,Y -126.9492,Z 179,A -111.6514,B 5.4432,C 0.3875,E1 5.3892,E2 204.1836} C_DIS
LIN {X -62.4894,Y -125.8416,Z 179,A -113.0609,B 5.4429,C 0.3905,E1 5.3856,E2 205.6427} C_DIS
LIN {X -65.8772,Y -124.1027,Z 179,A -114.3553,B 5.4433,C 0.3857,E1 5.3824,E2 206.9031} C_DIS
LIN {X -69.7609,Y -121.9627,Z 179,A -116.1354,B 5.4435,C 0.3831,E1 5.3781,E2 208.6796} C_DIS
LIN {X -73.4755,Y -119.7615,Z 179,A -117.8479,B 5.4437,C 0.3801,E1 5.374,E2 210.3856} C_DIS
LIN {X -76.9595,Y -117.5535,Z 179,A -119.6918,B 5.4437,C 0.3795,E1 5.3696,E2 212.251} C_DIS
LIN {X -80.4807,Y -115.1712,Z 179,A -121.2793,B 5.444,C 0.3753,E1 5.366,E2 213.819} C_DIS
LIN {X -85.7275,Y -111.3214,Z 179,A -124.1564,B 5.4441,C 0.3734,E1 5.3595,E2 216.7255} C_DIS
LIN {X -89.2741,Y -108.4979,Z 179,A -126.0468,B 5.4443,C 0.3707,E1 5.3554,E2 218.6212} C_DIS
LIN {X -92.7952,Y -105.5018,Z 179,A -127.946,B 5.4445,C 0.3675,E1 5.3514,E2 220.5218} C_DIS
LIN {X -96.1224,Y -102.4798,Z 179,A -129.8282,B 5.4447,C 0.3646,E1 5.3475,E2 222.4102} C_DIS
LIN {X -99.39,Y -99.3139,Z 179,A -131.7216,B 5.4449,C 0.3614,E1 5.3437,E2 224.3083} C_DIS
LIN {X -102.5361,Y -96.0624,Z 179,A -133.6035,B 5.4452,C 0.3581,E1 5.3401,E2 226.1945} C_DIS
LIN {X -105.5534,Y -92.7369,Z 179,A -135.459,B 5.4454,C 0.3546,E1 5.3367,E2 228.0528} C_DIS
LIN {X -108.4645,Y -89.3144,Z 179,A -137.3387,B 5.4456,C 0.3512,E1 5.3333,E2 229.9381} C_DIS
LIN {X -111.1554,Y -85.9416,Z 179,A -139.0448,B 5.4459,C 0.3468,E1 5.3303,E2 231.6366} C_DIS
LIN {X -113.8871,Y -82.2875,Z 179,A -141.0018,B 5.4461,C 0.3436,E1 5.3271,E2 233.6056} C_DIS
LIN {X -116.5227,Y -78.5111,Z 179,A -142.8959,B 5.4464,C 0.3394,E1 5.3241,E2 235.5012} C_DIS
LIN {X -119.5269,Y -73.8579,Z 179,A -145.6625,B 5.4464,C 0.339,E1 5.3199,E2 238.3329} C_DIS
LIN {X -121.8827,Y -69.9013,Z 179,A -147.5673,B 5.4466,C 0.3347,E1 5.3172,E2 240.2403} C_DIS
LIN {X -124.0573,Y -65.9637,Z 179,A -148.9705,B 5.4472,C 0.3261,E1 5.3154,E2 241.5867} C_DIS
LIN {X -125.8454,Y -62.4816,Z 179,A -150.5606,B 5.4474,C 0.322,E1 5.3134,E2 243.1753} C_DIS
LIN {X -127.2582,Y -59.5538,Z 179,A -152.051,B 5.4475,C 0.3202,E1 5.3116,E2 244.6865} C_DIS
LIN {X -129.0225,Y -55.6248,Z 179,A -153.6551,B 5.4479,C 0.3143,E1 5.3098,E2 246.2697} C_DIS
LIN {X -130.6346,Y -51.7287,Z 179,A -156.1973,B 5.4477,C 0.3175,E1 5.3071,E2 248.9175} C_DIS
LIN {X -132.5854,Y -46.5004,Z 179,A -157.8023,B 5.4484,C 0.3052,E1 5.3057,E2 250.4347} C_DIS
LIN {X -133.7078,Y -43.1664,Z 179,A -159.3239,B 5.4485,C 0.3022,E1 5.3043,E2 251.9667} C_DIS
LIN {X -134.6322,Y -40.1954,Z 179,A -160.7272,B 5.4487,C 0.3,E1 5.3032,E2 253.3867} C_DIS
LIN {X -135.7359,Y -36.2866,Z 179,A -162.2907,B 5.449,C 0.2946,E1 5.302,E2 254.9371} C_DIS
LIN {X -136.5228,Y -33.2049,Z 179,A -163.5691,B 5.4492,C 0.2909,E1 5.3012,E2 256.2123} C_DIS
LIN {X -137.3114,Y -29.7755,Z 179,A -165.1426,B 5.4492,C 0.2882,E1 5.3002,E2 257.8028} C_DIS
LIN {X -137.9982,Y -26.4098,Z 179,A -166.5381,B 5.4495,C 0.2842,E1 5.2995,E2 259.1966} C_DIS
LIN {X -138.6145,Y -22.9571,Z 179,A -168.0101,B 5.4497,C 0.2806,E1 5.2988,E2 260.6732} C_DIS
LIN {X -139.3431,Y -18.0157,Z 179,A -169.9851,B 5.45,C 0.2743,E1 5.298,E2 262.6388} C_DIS
LIN {X -139.9937,Y -11.9498,Z 179,A -172.6869,B 5.4503,C 0.2693,E1 5.2972,E2 265.3665} C_DIS
LIN {X -140.3639,Y -6.2425,Z 179,A -175.2541,B 5.4505,C 0.2648,E1 5.2968,E2 267.9621} C_DIS
LIN {X -140.4727,Y 2.984,Z 179,A -178.9074,B 5.451,C 0.2531,E1 5.2968,E2 271.5985} C_DIS
LIN {X -140.1171,Y 10.4046,Z 179,A 178.2967,B 5.4515,C 0.2423,E1 5.2972,E2 274.3622} C_DIS
LIN {X -139.4422,Y 17.2411,Z 179,A 175.1194,B 5.4517,C 0.2378,E1 5.2981,E2 277.5857} C_DIS
LIN {X -138.7826,Y 21.922,Z 179,A 173.1697,B 5.4519,C 0.2326,E1 5.2988,E2 279.5366} C_DIS
LIN {X -137.8399,Y 27.2323,Z 179,A 170.6934,B 5.4521,C 0.2289,E1 5.3001,E2 282.0464} C_DIS
LIN {X -137.0803,Y 30.8252,Z 179,A 169.2803,B 5.4523,C 0.224,E1 5.301,E2 283.4476} C_DIS
LIN {X -136.1843,Y 34.5657,Z 179,A 167.7172,B 5.4525,C 0.2196,E1 5.302,E2 285.0086} C_DIS
LIN {X -135.3228,Y 37.7981,Z 179,A 166.4568,B 5.4527,C 0.2149,E1 5.3029,E2 286.2547} C_DIS
LIN {X -134.388,Y 40.9978,Z 179,A 164.9241,B 5.4527,C 0.2127,E1 5.3041,E2 287.8082} C_DIS
LIN {X -133.404,Y 44.0955,Z 179,A 163.5408,B 5.4529,C 0.2097,E1 5.3053,E2 289.1978} C_DIS
LIN {X -132.0226,Y 48.0745,Z 179,A 161.7816,B 5.453,C 0.2054,E1 5.307,E2 290.9608} C_DIS
LIN {X -131.0272,Y 50.7232,Z 179,A 160.1853,B 5.453,C 0.2064,E1 5.3087,E2 292.612} C_DIS
LIN {X -129.5072,Y 54.4878,Z 179,A 158.8028,B 5.4532,C 0.1996,E1 5.3101,E2 293.9587} C_DIS
LIN {X -127.4218,Y 59.2,Z 179,A 156.7076,B 5.4534,C 0.194,E1 5.3125,E2 296.0513} C_DIS
LIN {X -126.2195,Y 61.7232,Z 179,A 154.838,B 5.4534,C 0.1978,E1 5.315,E2 298.0117} C_DIS
LIN {X -123.5255,Y 66.9556,Z 179,A 153.0163,B 5.4537,C 0.1865,E1 5.3172,E2 299.7588} C_DIS
LIN {X -121.3004,Y 70.9067,Z 179,A 151.1167,B 5.4538,C 0.1824,E1 5.3199,E2 301.6631} C_DIS
LIN {X -118.8831,Y 74.8885,Z 179,A 149.2087,B 5.454,C 0.1779,E1 5.3227,E2 303.5706} C_DIS
LIN {X -116.4609,Y 78.6025,Z 179,A 147.3749,B 5.4541,C 0.1738,E1 5.3255,E2 305.406} C_DIS
LIN {X -113.9883,Y 82.1479,Z 179,A 145.7181,B 5.4543,C 0.1687,E1 5.3281,E2 307.0479} C_DIS
LIN {X -111.9219,Y 84.9406,Z 179,A 143.9525,B 5.4543,C 0.1688,E1 5.3312,E2 308.8561} C_DIS
LIN {X -108.5711,Y 89.1846,Z 179,A 142.1236,B 5.4545,C 0.1603,E1 5.3343,E2 310.6358} C_DIS
LIN {X -105.0456,Y 93.3112,Z 179,A 138.9176,B 5.4544,C 0.1651,E1 5.3404,E2 313.9642} C_DIS
LIN {X -101.0408,Y 97.6332,Z 179,A 137.393,B 5.4548,C 0.1517,E1 5.3431,E2 315.377} C_DIS
LIN {X -96.2527,Y 102.3568,Z 179,A 134.5922,B 5.4549,C 0.1469,E1 5.3487,E2 318.183} C_DIS
LIN {X -90.5186,Y 107.4612,Z 179,A 131.3098,B 5.455,C 0.1425,E1 5.3556,E2 321.4821} C_DIS
LIN {X -87.1813,Y 110.1864,Z 179,A 129.4549,B 5.455,C 0.1404,E1 5.3597,E2 323.3478} C_DIS
LIN {X -82.51,Y 113.7259,Z 179,A 126.884,B 5.4551,C 0.1382,E1 5.3655,E2 325.9395} C_DIS
LIN {X -78.4156,Y 116.5874,Z 179,A 124.8746,B 5.4552,C 0.1347,E1 5.3701,E2 327.9439} C_DIS
LIN {X -74.593,Y 119.0694,Z 179,A 122.9582,B 5.4552,C 0.1325,E1 5.3746,E2 329.866} C_DIS
LIN {X -71.0513,Y 121.2155,Z 179,A 121.2605,B 5.4553,C 0.1301,E1 5.3787,E2 331.5635} C_DIS
LIN {X -67.1221,Y 123.4347,Z 179,A 119.4313,B 5.4554,C 0.1275,E1 5.3832,E2 333.39} C_DIS
LIN {X -64.2302,Y 124.9627,Z 179,A 118.1708,B 5.4554,C 0.125,E1 5.3863,E2 334.6403} C_DIS
Enddeposition()
END
